(* IEC 61131-3 sources: elnaProjects/ElpcLogic/PomarKc7Changed/FunctionBlocks (part 2) *)

(* ---- Если управление с ВУ заблокировано, то  передаем команду из алгоритма ---- *)
IF StrAlg.inOpcCommandsDisabled THEN
	StrAlg.inCommand := StrAlg.inCommand_Alg;
ELSE (* иначе передаем команду с АРМа*)
	StrAlg.inCommand := StrAlg.inCommand_ARM;
END_IF;

_sunpackerCommand(command := StrAlg.inCommand);
	source := _sunpackerCommand.source;
	cmd := _sunpackerCommand.cmd;

IF cmd <> 0 AND lastCmd <> cmd AND (((NOT StrAlg.opcCommandsDisabled) AND source > 0) OR source = 0) then
	CASE BYTE_TO_INT(cmd) OF
		(*cmdRun*) 1: 	IF (StrAlg.CanRun) THEN
					StrAlg.isRuning := TRUE;
					StrAlg.isEnded := FALSE;
					StrAlg.hasError := FALSE;
					(*****************       OnRun       *****************)

					cmd_for_Status := cmd;
					source_for_Status := source;
					command_error_for_Status := 0;
				ELSE
					StrAlg.isRuning := FALSE;
					StrAlg.isEnded := FALSE;
					StrAlg.hasError 	:= FALSE;

					cmd_for_Status := 0;
					source_for_Status := source;
					command_error_for_Status := cmd;
				END_IF;
		(*cmdReset*) 2: 	StrAlg.isRuning := FALSE;
				StrAlg.isEnded := FALSE;
				StrAlg.hasError 	:= FALSE;

                                         (*****************       OnReset       *****************)
                                        waitOn(in:=FALSE);
                                        waitOff(in:=FALSE);
                                        AlgTimers.AutoPns_OffTimer:=UDINT_TO_UINT(TIME_TO_UDINT(waitOff.pt -waitOff.ET)/1000);

				cmd_for_Status := cmd;
				source_for_Status := source;
				command_error_for_Status := 0;
	END_CASE;
	resetCmdTimer(IN := false);
	resetCmdTimerPriznak := TRUE;
END_IF;
lastCmd := cmd;

resetCmdTimer(IN := resetCmdTimerPriznak, PT := T#5S);
IF resetCmdTimer.Q THEN
	resetCmdTimerPriznak := FALSE;
	source_for_Status := 0;
	cmd_for_Status := 0;
	command_error_for_Status := 0;
END_IF;

(*TODO: TYPE PROGRAM CODE HERE*)
StrAlg.status :=  SHL(BYTE_TO_DWORD(source_for_Status), 29)
			OR SHL(BYTE_TO_DWORD(cmd_for_Status), 26)
			OR SHL(BYTE_TO_DWORD(command_error_for_Status), 23)
			OR SHL(BOOL_TO_DWORD(StrAlg.OpcCommandsDisabled ), 21)
			OR SHL(BOOL_TO_DWORD(StrAlg.hasError),4)
			OR SHL(BOOL_TO_DWORD(StrAlg.CanRun),2)
			OR SHL(BOOL_TO_DWORD(StrAlg.isEnded),1)
			OR BOOL_TO_DWORD(StrAlg.isRuning);

(* ---- fb_AutoTenAlg.st ---- *)
FUNCTION_BLOCK fb_AutoTenAlg

VAR_IN_OUT
	StrAlg : struct_Alg;
	PNS : struct_Switch;
	TEN : struct_Switch;
END_VAR

VAR_INPUT
	T_masla : struct_AI;
	Uroven_masla : struct_AI;
	offTemperature : struct_AnalogParametr;
END_VAR

VAR
	_sunpackerCommand : fb_sunpackerCommand;
	_statusAi : TYPE_StatusAi;
	_statusDualInput : TYPE_statusDualInput;
	_commandDualInput : TYPE_commandDualInput;
	source : BYTE;
	cmd : BYTE;
	lastCmd : BYTE;
	source_for_Status : BYTE;
	cmd_for_Status : BYTE;
	command_error_for_Status : BYTE;
	resetCmdTimer : TON;
	resetCmdTimerPriznak : BOOL;
	onInit : BOOL;
END_VAR

IF NOT onInit THEN
StrAlg.inCanRun:=TRUE;
onInit:=TRUE;
END_IF;

IF StrAlg.isRuning THEN

IF ((T_masla.interval >= _statusAi.normal) AND (T_masla.value > offTemperature.Value)) OR
((Uroven_masla.interval >= _statusAi.normal) AND (Uroven_masla.value < Uroven_masla.LA)) OR
(PNS.onStatus=_statusDualInput.STATUS_OFF) THEN

      TEN.inOpcCommandsDisabled:=TRUE;

	IF TEN.onStatus = _statusDualInput.STATUS_ON THEN
          TEN.inCommand_Alg:=BYTE_TO_WORD(_commandDualInput.CMD_OFF);
	END_IF;

ELSIF PNS.onStatus = _statusDualInput.STATUS_ON THEN
      TEN.inOpcCommandsDisabled:=FALSE;
END_IF;

END_IF;

StrAlg.CanRun := StrAlg.inCanRun;
StrAlg.hasError := TEN.CommandFault OR (T_masla.interval < _statusAi.normal) OR (Uroven_masla.interval < _statusAi.normal);

StrAlg.OpcCommandsDisabled := StrAlg.inOpcCommandsDisabled;

(* ---- Если управление с ВУ заблокировано, то  передаем команду из алгоритма ---- *)
IF StrAlg.inOpcCommandsDisabled THEN
	StrAlg.inCommand := StrAlg.inCommand_Alg;
ELSE (* иначе передаем команду с АРМа*)
	StrAlg.inCommand := StrAlg.inCommand_ARM;
END_IF;

_sunpackerCommand(command := StrAlg.inCommand);
	source := _sunpackerCommand.source;
	cmd := _sunpackerCommand.cmd;

IF cmd <> 0 AND lastCmd <> cmd AND (((NOT StrAlg.opcCommandsDisabled) AND source > 0) OR source = 0) then
	CASE BYTE_TO_INT(cmd) OF
		(*cmdRun*) 1: 	IF StrAlg.CanRun AND NOT StrAlg.hasError THEN
					StrAlg.isRuning := TRUE;
					StrAlg.isEnded := FALSE;
					(*StrAlg.hasError := FALSE;*)

                                                  (*****************       OnRun       *****************)
                                                  IF StrAlg.inOpcCommandsDisabled THEN
		                              StrAlg.inOpcCommandsDisabled:=FALSE;
                                                  END_IF;
					cmd_for_Status := cmd;
					source_for_Status := source;
					command_error_for_Status := 0;
				ELSE
					StrAlg.isRuning := FALSE;
					StrAlg.isEnded := FALSE;
					(*StrAlg.hasError 	:= FALSE;*)

					cmd_for_Status := 0;
					source_for_Status := source;
					command_error_for_Status := cmd;
				END_IF;
		(*cmdReset*) 2: 	StrAlg.isRuning := FALSE;
				StrAlg.isEnded := FALSE;
				(*StrAlg.hasError 	:= FALSE;*)

                                        (*****************       OnReset       *****************)
                                        TEN.inOpcCommandsDisabled:=TRUE;
                                        TEN.inCommand_Alg:=BYTE_TO_WORD(_commandDualInput.CMD_OFF);

				cmd_for_Status := cmd;
				source_for_Status := source;
				command_error_for_Status := 0;
	END_CASE;
	resetCmdTimer(IN := false);
	resetCmdTimerPriznak := TRUE;
END_IF;
lastCmd := cmd;

resetCmdTimer(IN := resetCmdTimerPriznak, PT := T#5S);
IF resetCmdTimer.Q THEN
	resetCmdTimerPriznak := FALSE;
	source_for_Status := 0;
	cmd_for_Status := 0;
	command_error_for_Status := 0;
END_IF;

(*TODO: TYPE PROGRAM CODE HERE*)
StrAlg.status :=  SHL(BYTE_TO_DWORD(source_for_Status), 29)
			OR SHL(BYTE_TO_DWORD(cmd_for_Status), 26)
			OR SHL(BYTE_TO_DWORD(command_error_for_Status), 23)
			OR SHL(BOOL_TO_DWORD(StrAlg.OpcCommandsDisabled ), 21)
			OR SHL(BOOL_TO_DWORD(StrAlg.hasError),4)
			OR SHL(BOOL_TO_DWORD(StrAlg.CanRun),2)
			OR SHL(BOOL_TO_DWORD(StrAlg.isEnded),1)
			OR BOOL_TO_DWORD(StrAlg.isRuning);

(* ---- fb_BaseAlgoritm.st ---- *)
FUNCTION_BLOCK fb_BaseAlgoritm

VAR_IN_OUT
	StrAlg : struct_Alg;
END_VAR

VAR
	_sunpackerCommand : fb_sunpackerCommand;
	source : BYTE;
	cmd : BYTE;
	lastCmd : BYTE;
	source_for_Status : BYTE;
	cmd_for_Status : BYTE;
	command_error_for_Status : BYTE;
	resetCmdTimer : TON;
	resetCmdTimerPriznak : BOOL;
END_VAR

StrAlg.CanRun := StrAlg.inCanRun;
StrAlg.hasError := StrAlg.inHasError OR (command_error_for_Status <> 0);
StrAlg.isEnded := StrAlg.inEnded;

StrAlg.OpcCommandsDisabled := StrAlg.inOpcCommandsDisabled;

(* ---- Если управление с ВУ заблокировано, то передаем команду из алгоритма ---- *)
IF StrAlg.inOpcCommandsDisabled THEN
	StrAlg.inCommand := StrAlg.inCommand_Alg;
ELSE (* иначе передаем команду с АРМа*)
	StrAlg.inCommand := StrAlg.inCommand_ARM;
END_IF;

_sunpackerCommand(command := StrAlg.inCommand);
	source := _sunpackerCommand.source;
	cmd := _sunpackerCommand.cmd;

IF cmd <> 0 AND lastCmd <> cmd AND (((NOT StrAlg.opcCommandsDisabled) AND source > 0) OR source = 0) then
	CASE BYTE_TO_INT(cmd) OF
		(*cmdRun*) 1: 	IF (StrAlg.CanRun) THEN
					StrAlg.isRuning := TRUE;
					StrAlg.isEnded := FALSE;
					StrAlg.hasError 	:= FALSE;

					cmd_for_Status := cmd;
					source_for_Status := source;
					command_error_for_Status := 0;
				ELSE
					StrAlg.isRuning := FALSE;
					StrAlg.isEnded := FALSE;
					StrAlg.hasError 	:= FALSE;

					cmd_for_Status := 0;
					source_for_Status := source;
					command_error_for_Status := cmd;
				END_IF;
		(*cmdReset*) 2: 	StrAlg.isRuning := FALSE;
				StrAlg.isEnded := FALSE;
				StrAlg.hasError 	:= FALSE;
				cmd_for_Status := cmd;
				source_for_Status := source;
				command_error_for_Status := 0;
	END_CASE;
	resetCmdTimer(IN := false);
	resetCmdTimerPriznak := TRUE;
END_IF;
lastCmd := cmd;

resetCmdTimer(IN := resetCmdTimerPriznak, PT := T#5S);
IF resetCmdTimer.Q THEN
	resetCmdTimerPriznak := FALSE;
	source_for_Status := 0;
	cmd_for_Status := 0;
	command_error_for_Status := 0;
END_IF;

StrAlg.status :=  SHL(BYTE_TO_DWORD(source_for_Status), 29)
			OR SHL(BYTE_TO_DWORD(cmd_for_Status), 26)
			OR SHL(BYTE_TO_DWORD(command_error_for_Status), 23)
			OR SHL(BOOL_TO_DWORD(StrAlg.OpcCommandsDisabled ), 21)
			OR SHL(BOOL_TO_DWORD(StrAlg.hasError),4)
			OR SHL(BOOL_TO_DWORD(StrAlg.CanRun),2)
			OR SHL(BOOL_TO_DWORD(StrAlg.isEnded),1)
			OR BOOL_TO_DWORD(StrAlg.isRuning);

(* ---- fb_BaseProtection.st ---- *)
FUNCTION_BLOCK fb_BaseProtection

VAR_INPUT
	inSignaling : BOOL;
	inTag : BYTE;
	inRunOnStart : BOOL;
	inCanRun : BOOL;
	inHasError : BOOL;
	inEnded : BOOL;
	inOpcCommandsDisabled : BOOL;
	inCommand : WORD;
END_VAR

VAR_OUTPUT
	Tag : BYTE;
	status : DWORD;
	CanRun : BOOL;
	OpcCommandsDisabled : BOOL;
	isRunning : BOOL;
	HasError : BOOL;
	isEnded : BOOL;
	Remont : BOOL;
	Check : BOOL;
	Signaling : BOOL;
	SignalingTP : BOOL;
	RunOnStart : BOOL;
END_VAR

VAR
	_sunpackerCommand : fb_sunpackerCommand;
	_ProtectionTags : TYPE_ProtectionTags;
	_signalingTp : TOF;
	source : BYTE;
	cmd : BYTE;
	lastCmd : BYTE;
	source_for_Status : BYTE;
	cmd_for_Status : BYTE;
	command_error_for_Status : BYTE;
	resetCmdTimer : TON;
	resetCmdTimerPriznak : BOOL;
	signalinTimer : TON;
	runOnStart_Trig : R_TRIG;
END_VAR

Tag := inTag;
RunOnStart := inRunOnStart;

CanRun := inCanRun;
hasError := inHasError;
isEnded := inEnded;

OpcCommandsDisabled := inOpcCommandsDisabled;

_sunpackerCommand(command := inCommand);
	source := _sunpackerCommand.source;
	cmd := _sunpackerCommand.cmd;

IF cmd <> 0 AND lastCmd <> cmd AND (((NOT opcCommandsDisabled) AND source > 0) OR source = 0) then
	CASE BYTE_TO_INT(cmd) OF
		(*cmdRun*) 1: 	IF CanRun AND NOT Remont THEN
					isEnded := FALSE;
					hasError 	:= FALSE;
					isRunning := TRUE;
					cmd_for_Status := cmd;
					source_for_Status := source;
					command_error_for_Status := 0;
				ELSE
					isRunning := FALSE;
					isEnded := FALSE;
					hasError 	:= FALSE;

					cmd_for_Status := 0;
					source_for_Status := source;
					command_error_for_Status := cmd;
				END_IF;
		(*cmdReset*) 2: 	isRunning := FALSE;
				isEnded := FALSE;
				hasError 	:= FALSE;
				inSignaling := FALSE;
				Check := FALSE;
				cmd_for_Status := cmd;
				source_for_Status := source;
				command_error_for_Status := 0;
	(*cmd_setRemont*) 4 :	Remont := TRUE;
				isRunning := FALSE;

				cmd_for_Status := cmd;
				source_for_Status := source;
				command_error_for_Status := 0;
	(*cmd_resetRemont*) 5 : 	IF inSignaling THEN
					cmd_for_Status := 0;
					source_for_Status := 0;
					command_error_for_Status := cmd;
				ELSE
					Remont := FALSE;
					isRunning := TRUE;

					cmd_for_Status := cmd;
					source_for_Status := source;
					command_error_for_Status := 0;
				END_IF;
	(*cmd_setCheck*) 6 : 	Check := TRUE;

				cmd_for_Status := cmd;
				source_for_Status := source;
				command_error_for_Status := 0;
	END_CASE;
	resetCmdTimer(IN := false);
	resetCmdTimerPriznak := TRUE;
END_IF;
lastCmd := cmd;

resetCmdTimer(IN := resetCmdTimerPriznak);
IF resetCmdTimer.Q THEN
	resetCmdTimerPriznak := FALSE;
	source_for_Status := 0;
	cmd_for_Status := 0;
	command_error_for_Status := 0;
END_IF;

IF isRunning THEN
	Signaling := inSignaling;
	SignalingTP := _signalingTp.Q;
ELSE
	Signaling := 0;
	SignalingTP := 0;
END_IF;

IF NOT Remont AND NOT Check THEN
	_signalingTp(in := Signaling, PT := T#1s);
ELSE
	_signalingTp(in := FALSE);
END_IF;

status :=  SHL(BYTE_TO_DWORD(source_for_Status), 29)
			OR SHL(BYTE_TO_DWORD(cmd_for_Status), 26)
			OR SHL(BYTE_TO_DWORD(command_error_for_Status), 23)
			OR SHL(BOOL_TO_DWORD(OpcCommandsDisabled ), 21)
			OR SHL(BOOL_TO_DWORD(Signaling), 16)
			OR SHL(BOOL_TO_DWORD(RunOnStart ), 15)
			OR SHL(BOOL_TO_DWORD(remont), 6)
			OR SHL(BOOL_TO_DWORD(Check), 5)
			OR SHL(BOOL_TO_DWORD(hasError), 4)
			OR SHL(BOOL_TO_DWORD(SignalingTP), 3)
			OR SHL(BOOL_TO_DWORD(CanRun), 2)
			OR SHL(BOOL_TO_DWORD(isEnded), 1)
			OR BOOL_TO_DWORD(isRunning);

(* ---- fb_DI_Init.st ---- *)
FUNCTION_BLOCK fb_DI_Init

VAR_INPUT
	data_Ini : BOOL; (*Флаг необходимости инициализации параметров.*)
	imit : BOOL          := FALSE;
END_VAR

VAR_IN_OUT
	strDI : struct_DI;
END_VAR

VAR_OUTPUT
	Init : BOOL          := FALSE; (*Флаг успешно выполненной инициализации.*)
END_VAR

(*****            Функциональный блок переинициализации структуры-дескриптора канала дискретного ввода        *****)

 Init := FALSE;

    IF data_Ini THEN                            (* Параметрам требуется переинициализация. *)
        strDI.imit       := imit;
        data_Ini:=FALSE;
        Init := TRUE;
    END_IF;
  IF Init THEN
imit:=FALSE;
    END_IF;

(* ---- fb_DiProtection.st ---- *)
FUNCTION_BLOCK fb_DiProtection

VAR_INPUT
	di : struct_singleSignal;
END_VAR

VAR_IN_OUT
	StrDIp : struct_DiProtection;
END_VAR

VAR
	_sunpackerCommand : fb_sunpackerCommand;
	_ProtectionTags : TYPE_ProtectionTags;
	_signalingTp : TOF;
	timer : TON;
	SignalingTrig : R_TRIG;
	SignalingFTrig : F_TRIG;
	SignalingDi : BOOL;
	source : BYTE;
	cmd : BYTE;
	lastCmd : BYTE;
	source_for_Status : BYTE;
	cmd_for_Status : BYTE;
	command_error_for_Status : BYTE;
	resetCmdTimer : TON;
	resetCmdTimerPriznak : BOOL;
	signalinTimer : TON;
	runOnStart_Trig : R_TRIG;
END_VAR

timer(IN := di.Q AND StrDIp.isRunning  , PT := StrDIp.delay);
SignalingTrig(CLK := timer.Q);
IF SignalingTrig.Q THEN
	SignalingDi := TRUE;
END_IF;
SignalingFTrig(CLK := timer.Q);
IF SignalingFTrig.Q THEN
	SignalingDi := FALSE;
END_IF;

StrDIp.Tag := StrDIp.inTag;
StrDIp.RunOnStart := StrDIp.inRunOnStart;

StrDIp.CanRun := StrDIp.inCanRun;

StrDIp.OpcCommandsDisabled := StrDIp.inOpcCommandsDisabled;

(* ---- Если управление с ВУ заблокировано, то передаем команду из алгоритма ---- *)
IF StrDIp.inOpcCommandsDisabled THEN
	StrDIp.inCommand := StrDIp.inCommand_Alg;
ELSE (* иначе передаем команду с АРМа*)
	StrDIp.inCommand := StrDIp.inCommand_ARM;
END_IF;

_sunpackerCommand(command := StrDIp.inCommand);
	source := _sunpackerCommand.source;
	cmd := _sunpackerCommand.cmd;

IF cmd <> 0 AND lastCmd <> cmd AND (((NOT StrDIp.opcCommandsDisabled) AND source > 0) OR source = 0) then

	CASE BYTE_TO_INT(cmd) OF
	        (*cmdRun*) 1: 	IF        NOT StrDIp.Remont THEN
					StrDIp.isEnded := FALSE;
					StrDIp.hasError 	:= FALSE;
					StrDIp.isRunning := TRUE;
					cmd_for_Status := cmd;
					source_for_Status := source;
					command_error_for_Status := 0;
				ELSE
					StrDIp.isRunning := FALSE;
					StrDIp.isEnded := FALSE;
					StrDIp.hasError 	:= FALSE;

					cmd_for_Status := 0;
					source_for_Status := source;
					command_error_for_Status := cmd;
				END_IF;
                                        StrDIp.inOpcCommandsDisabled:=FALSE;

                (*cmdReset*) 2: 	StrDIp.isRunning := FALSE;
				StrDIp.isEnded := FALSE;
				StrDIp.hasError 	:= FALSE;
				SignalingDi:= FALSE;
				StrDIp.Check := FALSE;
				cmd_for_Status := cmd;
				source_for_Status := source;
				command_error_for_Status := 0;
                                       StrDIp.inOpcCommandsDisabled:=FALSE;

	(*cmd_setRemont*) 4 :	StrDIp.Remont := TRUE;
				(*StrDIp.isRunning := FALSE;*)

				cmd_for_Status := cmd;
				source_for_Status := source;
				command_error_for_Status := 0;
        (*cmd_resetRemont*) 5 : 	(*IF di.Q THEN
					cmd_for_Status := 0;
					source_for_Status := 0;
					command_error_for_Status := cmd;
				ELSE*)
					StrDIp.Remont := FALSE;
					(*StrDIp.isRunning := TRUE;*)

					cmd_for_Status := cmd;
					source_for_Status := source;
					command_error_for_Status := 0;
				(*END_IF;*)
	(*cmd_setCheck*) 6 : 	StrDIp.Check := TRUE;

				cmd_for_Status := cmd;
				source_for_Status := source;
				command_error_for_Status := 0;
	END_CASE;
	resetCmdTimer(IN := false);
	resetCmdTimerPriznak := TRUE;
END_IF;
lastCmd := cmd;

resetCmdTimer(IN := resetCmdTimerPriznak);
IF resetCmdTimer.Q THEN
	resetCmdTimerPriznak := FALSE;
	source_for_Status := 0;
	cmd_for_Status := 0;
	command_error_for_Status := 0;
END_IF;

IF StrDIp.isRunning AND NOT StrDIp.Remont AND NOT StrDIp.Check THEN
	StrDIp.Signaling := SignalingDi;
	StrDIp.SignalingTP := _signalingTp.Q;
ELSE
	StrDIp.Signaling := 0;
	StrDIp.SignalingTP := 0;
END_IF;

_signalingTp(in := StrDIp.Signaling, PT := T#1s);

StrDIp.status :=  SHL(BYTE_TO_DWORD(source_for_Status), 29)
			OR SHL(BYTE_TO_DWORD(cmd_for_Status), 26)
			OR SHL(BYTE_TO_DWORD(command_error_for_Status), 23)
			OR SHL(BOOL_TO_DWORD(StrDIp.OpcCommandsDisabled ), 21)
			OR SHL(BOOL_TO_DWORD(StrDIp.Signaling), 16)
			OR SHL(BOOL_TO_DWORD(StrDIp.RunOnStart ), 15)
			OR SHL(BOOL_TO_DWORD(StrDIp.remont), 6)
			OR SHL(BOOL_TO_DWORD(StrDIp.Check), 5)
			OR SHL(BOOL_TO_DWORD(StrDIp.hasError), 4)
			OR SHL(BOOL_TO_DWORD(StrDIp.SignalingTP), 3)
			OR SHL(BOOL_TO_DWORD(StrDIp.CanRun), 2)
			OR SHL(BOOL_TO_DWORD(StrDIp.isEnded), 1)
			OR BOOL_TO_DWORD(StrDIp.isRunning);

(* ---- fb_DiProtection_Init.st ---- *)
FUNCTION_BLOCK fb_DiProtection_Init

VAR_INPUT
	data_Ini : BOOL; (*Флаг необходимости инициализации параметров.*)
	delay : TIME;
	inTag : BYTE;
	inRunOnStart : BOOL;
END_VAR

VAR_IN_OUT
	str_DIp : struct_DiProtection;
END_VAR

VAR_OUTPUT
	Init : BOOL          := FALSE; (*Флаг успешно выполненной инициализации.*)
END_VAR

(*****            Функциональный блок переинициализации структуры  AiProtection          *****)

 Init := FALSE;

    IF data_Ini THEN                            (* Параметрам требуется переинициализация. *)
        str_DIp.delay               := delay;
        str_DIp.inTag               := inTag;
        str_DIp.inRunOnStart        := inRunOnStart;

        data_Ini:=FALSE;
        Init := TRUE;
    END_IF;
    IF Init THEN
        delay:= T#0S;
        inTag:= 0;
        inRunOnStart:= FALSE;
    END_IF;

(* ---- fb_DiscretParametr.st ---- *)
FUNCTION_BLOCK fb_DiscretParametr

VAR_IN_OUT
	StrDP : struct_DiscretParametr;
END_VAR

VAR
	_sunpackerCommand : fb_sunpackerCommand;
	source : BYTE;
	cmd : BYTE;
	parametr : BYTE;
	lastParametr : BYTE;
	source_for_Status : BYTE;
	cmd_for_Status : BYTE;
	command_error_for_Status : BYTE;
	resetCmdTimer : TON;
	resetCmdTimerPriznak : BOOL;
	secondTact : BOOL;
END_VAR

IF NOT secondTact THEN
	StrDP.Value := StrDP.currentValue;
	secondTact := true;
END_IF;

StrDP.OpcCommandsDisabled := StrDP.inOpcCommandsDisabled;

(* ---- Если управление с ВУ заблокировано, то передаем команду из алгоритма ---- *)
IF StrDP.inOpcCommandsDisabled THEN
	StrDP.inCommand := StrDP.inCommand_Alg;
ELSE (* иначе передаем команду с АРМа*)
	StrDP.inCommand := StrDP.inCommand_ARM;
END_IF;

_sunpackerCommand(command := StrDP.inCommand);
	source := _sunpackerCommand.source;
          parametr := _sunpackerCommand.parametr;
	cmd := _sunpackerCommand.cmd;

IF NOT StrDP.inOpcCommandsDisabled THEN
StrDP.newValue:= BYTE_TO_UINT(parametr);
END_IF;

IF cmd <> 0 AND StrDP.Value <> StrDP.newValue AND (((NOT StrDP.opcCommandsDisabled) AND source > 0) OR source = 0) then
	CASE BYTE_TO_INT(cmd) OF
	(*cmd_ChangeValue*) 1 :
                                  StrDP.Value := StrDP.newValue;
                                  StrDP.opcCommandsDisabled:=FALSE;
	END_CASE;
	source_for_Status := source;
	cmd_for_Status := cmd;
	resetCmdTimer(IN := FALSE);
	resetCmdTimerPriznak := TRUE;
END_IF;

lastParametr := parametr;

StrDP.status := SHL(BYTE_TO_DWORD(source_for_Status), 29)
			OR SHL(BYTE_TO_DWORD(cmd_for_Status), 26)
			OR SHL(BYTE_TO_DWORD(command_error_for_Status), 23)
			OR SHL(BOOL_TO_DWORD(StrDP.OpcCommandsDisabled ), 21)
                              OR SHL(UINT_TO_DWORD(StrDP.Value), 5);

resetCmdTimer(IN := resetCmdTimerPriznak, PT := T#5S);
IF resetCmdTimer.Q THEN
	resetCmdTimerPriznak := FALSE;
	source_for_Status := 0;
	cmd_for_Status := 0;
	command_error_for_Status := 0;
END_IF;

(* ---- fb_DiscretParametr_Init.st ---- *)
FUNCTION_BLOCK fb_DiscretParametr_Init

VAR_INPUT
	data_Ini : BOOL; (*Флаг необходимости инициализации параметров.*)
	currentValue : UINT;
END_VAR

VAR_IN_OUT
	strDp : struct_DiscretParametr;
END_VAR

VAR_OUTPUT
	Init : BOOL          := FALSE; (*Флаг успешно выполненной инициализации.*)
END_VAR

(*****            Функциональный блок переинициализации дискретного параметра.          *****)

 Init := FALSE;

    IF data_Ini THEN                            (* Параметрам требуется переинициализация. *)
        strDp.currentValue       := currentValue;
        data_Ini:=FALSE;
        Init := TRUE;
    END_IF;
IF Init THEN
currentValue:=0;
END_IF;

(* ---- fb_DiSourceMlp.st ---- *)
FUNCTION_BLOCK fb_DiSourceMlp

VAR_INPUT
	arDIN : TItemDIN;
	err_mod : TItemDIN;
END_VAR

VAR_IN_OUT
	strDI : struct_DI;
END_VAR

VAR_OUTPUT
	Bounce : BOOL; (*Дребезг контактов*)
END_VAR

VAR
	_value : WORD;
	_reliability : BOOL;
	bitNumber : INT;
	bitNum : INT;
END_VAR

strDI.blConnect := (*((UINT_TO_WORD(arDIN.wFlags) = 1472) and*) (UINT_TO_WORD(err_mod.wValue) = 20) and (UINT_TO_WORD(err_mod.wFlags) = 192);
Bounce := (UINT_TO_WORD(arDIN.wFlags) AND 16#0020) <> 0;

If NOT strDI.imit THEN
_value:=UINT_TO_WORD(arDIN.wValue);

    IF strDI.blConnect THEN
          strDI.reliability:=0;
          strDI.value:=0;
	FOR bitNumber:=0 TO 7 BY 1 DO

		_reliability:=WORD_TO_BOOL(SHR(_value, bitNumber*2) AND 16#2);
		strDI.reliability:=strDI.reliability OR SHL(BOOL_TO_WORD(_reliability),bitNumber);
		IF _reliability THEN
			strDI.value:=strDI.value OR SHL((SHR(_value, bitNumber*2) AND 16#1),bitNumber);
		END_IF;
	END_FOR;
    ELSE
	strDI.reliability := 0;
    END_IF;

    FOR bitNum:=0 TO 15 BY 1 DO
	          strDI.bits[bitNum].reliability :=WORD_TO_BOOL(SHR(strDI.reliability, bitNum) AND 16#1);
	IF strDI.bits[bitNum].reliability THEN
		strDI.bits[bitNum].value :=WORD_TO_BOOL(SHR(strDI.value, bitNum) AND 16#1);
                    strDI.bits[bitNum]._inversed :=NOT strDI.bits[bitNum].value;
	END_IF;
    END_FOR;

END_IF;

(* ---- fb_DO_Init.st ---- *)
FUNCTION_BLOCK fb_DO_Init

VAR_INPUT
	data_Ini : BOOL; (*Флаг необходимости инициализации параметров.*)
	imit : BOOL          := FALSE; (*Действие при неисправности канала AI.*)
END_VAR

VAR_IN_OUT
	strDO : struct_DO; (*Дескриптор DO-канала.*)
END_VAR

VAR_OUTPUT
	Init : BOOL          := FALSE; (*Флаг успешно выполненной инициализации.*)
END_VAR

(*****            Функциональный блок переинициализации структуры-дескриптора канала дискретного ввода.            *****)
 Init := FALSE;

    IF data_Ini THEN                            (* Параметрам требуется переинициализация. *)
        strDO.imit       := imit;
        data_Ini:=FALSE;
        Init := TRUE;
    END_IF;
  IF Init THEN
imit:=FALSE;
   END_IF;

(* ---- fb_DOSourceMlp.st ---- *)
FUNCTION_BLOCK fb_DOSourceMlp

VAR_IN_OUT
	arDout : TWordData; (*Данные для модуля DO.*)
END_VAR

VAR_INPUT
	err_mod : TItemDIN;
END_VAR

VAR_IN_OUT
	strDO : struct_DO; (*Текущие параметры канала DO.*)
END_VAR

VAR
	bitNumber : INT;
END_VAR

strDO.blConnect := ((UINT_TO_WORD(err_mod.wValue) = 20) and (UINT_TO_WORD(err_mod.wFlags) = 192));

strDO.value:=0;

FOR bitNumber:=0 TO 15 BY 1 DO
	strDO.value:=strDO.value OR (SHL(BOOL_TO_WORD(strDO.bits[bitNumber]),bitNumber));
END_FOR;

IF NOT strDO.imit THEN
	 arDout.wValue:= WORD_TO_UINT(strDO.value);
END_IF;

(* ---- fb_DualStateIm.st ---- *)
FUNCTION_BLOCK fb_DualStateIm

VAR_INPUT
	statOn : BOOL;
	statOff : BOOL;
END_VAR

VAR_IN_OUT
	StrDs : struct_DualStateIm;
END_VAR

VAR_INPUT
	statOn_reliability : BOOL;
	statOff_reliability : BOOL;
	inNs : TYPE_ReliableBit;
	inAccident : TYPE_ReliableBit;
	inCommand : WORD;
END_VAR

VAR
	_statOn : BOOL;
	_statOff : BOOL;
	getSdvig : BOOL;
	lastOnStatus : BYTE;
	cmd : BYTE;
	source : BYTE;
	lastCmd : BYTE;
	source_for_Status : BYTE;
	cmd_for_Status : BYTE;
	command_error_for_Status : BYTE;
	_sunpackerCommand : fb_sunpackerCommand;
	_statusDualInput : TYPE_statusDualInput;
	_commandDualInput : TYPE_commandDualInput;
	_commandErrorTimer : BOOL;
	onInit : BOOL          := FALSE;
	resetErrorTimer : BOOL;
	_changWithoutCommand : BOOL;
	errorCMDTimer : TON;
	sdvigReset : TON;
	_errorReset : TON;
END_VAR

VAR_IN_OUT
	cmdOn : BOOL;
END_VAR

VAR_OUTPUT
	cmdOff : BOOL;
END_VAR

IF NOT onInit THEN
IF StrDs.ISVALIDREF_cmdOn XOR StrDs.ISVALIDREF_cmdOff THEN
	IF 	StrDs.ISVALIDREF_cmdOn THEN
		lastCmd:= 2; (*baseCmdOff*)
	ELSE
		lastCmd:= 1; (*baseCmdOn*)
	END_IF;
END_IF;
onInit:=TRUE;
END_IF;

(* ---- Если управление с ВУ заблокировано, то в ИМ передаем команду из алгоритма ---- *)
IF StrDs.inOpcCommandsDisabled THEN
	StrDs.inCommand := StrDs.inCommand_Alg;
ELSE (* иначе передаем команду с АРМа*)
	StrDs.inCommand := StrDs.inCommand_ARM;
END_IF;

(* ---- Формирование состояния механизма ---- *)

IF (StrDs.ISVALIDREF_statOn) OR (StrDs.ISVALIDREF_statOff) THEN
	IF (StrDs.ISVALIDREF_statOn) AND (StrDs.ISVALIDREF_statOff) THEN
	StrDs.reliability:= statOn_reliability AND statOff_reliability;
		_statOn  := statOn;
		_statOff := statOff;
	ELSIF (StrDs.ISVALIDREF_statOn) THEN
                     StrDs.reliability:= statOn_reliability;
		_statOn  := statOn;
		_statOff := NOT statOn;
	ELSIF (StrDs.ISVALIDREF_statOff) THEN
		 StrDs.reliability:= statOff_reliability;
		_statOn  := NOT statOff;
		_statOff :=statOff;
	END_IF;

	IF StrDs.reliability THEN
		IF _statOn AND NOT _statOff 		THEN 	StrDs.onStatus := _statusDualInput.STATUS_ON;
		ELSIF _statOff AND NOT _statOn 	THEN 	StrDs.onStatus := _statusDualInput.Status_OFF;
		ELSIF NOT _statOn AND NOT _statOff 	THEN 	StrDs.onStatus := _statusDualInput.STATUS_TRANSITIONAL;
		ELSE					StrDs.onStatus := _statusDualInput.STATUS_ERROR;
                    END_IF;

	ELSE
		StrDs.onStatus := _statusDualInput.STATUS_NOTDEFINED;

	END_IF;
ELSE
	CASE BYTE_TO_INT(lastCmd) OF
		(*baseCmdOn*) 1: StrDs.onStatus  := _statusDualInput.STATUS_ON;
		(*baseCmdOff*) 2: StrDs.onStatus  := _statusDualInput.STATUS_OFF;

	ELSE
		 StrDs.onStatus := _statusDualInput.STATUS_NOTDEFINED;

	END_CASE;
END_IF;

(* ---- Формирование признака сдвига ---- *)
getSdvig := FALSE;
IF (StrDs.ISVALIDREF_cmdOn OR StrDs.ISVALIDREF_cmdOff) THEN
	IF NOT (StrDs.CmdOn OR StrDs.CmdOff) THEN
                     IF (lastOnStatus <> StrDs.onStatus AND
		(StrDs.onStatus <> _statusDualInput.STATUS_NOTDEFINED AND
                     StrDs.onStatus <> _statusDualInput.STATUS_ERROR)     AND
		(lastOnStatus <> _statusDualInput.STATUS_NOTDEFINED   AND
                     lastOnStatus <> _statusDualInput.STATUS_ERROR))
                    THEN
			getSdvig   := TRUE;
		END_IF;
	END_IF;
END_IF;

IF getSdvig THEN StrDs.sdvig:= TRUE; END_IF;

sdvigReset(IN:=StrDs.sdvig, PT:=T#15S);

IF sdvigReset.Q THEN StrDs.sdvig:=FALSE; END_IF;

lastOnStatus := StrDs.onStatus;

StrDs.Accident := inAccident.value AND inAccident.reliability;
StrDs.Ns := inNs.value AND inNs.reliability;
StrDs.OpcCommandsDisabled := StrDs.inOpcCommandsDisabled;

(* ---- Распаковка команды ---- *)
_sunpackerCommand(command := StrDs.inCommand);
	cmd := _sunpackerCommand.cmd;
	source := _sunpackerCommand.source;

(* ---- Обработка команды ---- *)
IF cmd <> 0 AND lastCmd <> cmd and (((NOT StrDs.opcCommandsDisabled) AND source > 0) OR source = 0) then
	CASE BYTE_TO_INT(cmd) OF
	(*cmd_open*) 1 :
			IF  StrDs.ISVALIDREF_cmdOn THEN StrDs.CmdOn := TRUE;
				IF StrDs.ISVALIDREF_cmdOff THEN StrDs.CmdOff := FALSE; END_IF;
			ELSIF  StrDs.ISVALIDREF_cmdOff THEN StrDs.CmdOff := FALSE;  END_IF;
			errorCMDTimer(IN := false);
			_commandErrorTimer := true;
			StrDs.lastCmdIsOn := true;
	(*cmd_close*) 2 :
			IF StrDs.ISVALIDREF_cmdOff THEN StrDs.CmdOff := TRUE;
				IF StrDs.ISVALIDREF_cmdOn THEN StrDs.CmdOn := FALSE; END_IF;
			ELSIF StrDs.ISVALIDREF_cmdOn THEN StrDs.CmdOn := FALSE; END_IF;
			errorCMDTimer(IN := false);
			_commandErrorTimer := true;
			StrDs.lastCmdIsOn := false;
	(*cmd_reset*) 3 :    IF StrDs.ISVALIDREF_statOn OR StrDs.ISVALIDREF_statOff THEN
			StrDs.CmdOn := FALSE;
			StrDs.CmdOff := FALSE;
                              lastCmd :=0;
			_commandErrorTimer := false;
			StrDs.lastCmdIsOn := false;
                              END_IF;
	END_CASE;
	source_for_Status := source;
	cmd_for_Status := cmd;
	command_error_for_Status := 0;
END_IF;

lastCmd := cmd;
errorCMDTimer(In := _commandErrorTimer, PT :=T#10s);

(* ---- алгоритм  для команды ВКЛючить ---- *)
IF (StrDs.onStatus = _statusDualInput.STATUS_ON) and (lastCmd = _commandDualInput.CMD_ON) then
	IF StrDs.ISVALIDREF_cmdOn AND StrDs.ISVALIDREF_cmdOff then  StrDs.cmdOn := false; END_IF;

	 errorCMDTimer(In := false);
	 _commandErrorTimer := false;
	 cmd_for_Status := 0;
	 source_for_Status := 0;
END_IF;

(* ---- off ---- *)
IF (StrDs.onStatus = _statusDualInput.STATUS_OFF) and (lastCmd = _commandDualInput.CMD_OFF) then
	IF StrDs.ISVALIDREF_cmdOn AND StrDs.ISVALIDREF_cmdOff then  StrDs.cmdOff := false; END_IF;

	 errorCMDTimer(In := false);
	 _commandErrorTimer := false;
	 cmd_for_Status := 0;
	 source_for_Status := 0;
END_IF;

(* ---- ошибка исполнения команды ---- *)
if errorCMDTimer.Q and (cmd_for_Status <> 0) then
	command_error_for_Status :=  cmd_for_Status;
	_commandErrorTimer := false;
	StrDs.CmdOn := false;
	StrDs.CmdOff := false;
	lastCmd := 0;
end_if;

(* ---- сброс ошибки команды ---- *)
StrDs.CommandFault := command_error_for_Status <> 0;
_errorReset(IN := command_error_for_Status <> 0, PT := T#15S);
IF _errorReset.Q THEN
	cmd_for_Status := 0;
	source_for_Status := 0;
	command_error_for_Status := 0;
END_IF;

cmdOn := StrDs.cmdOn;
cmdOff:= StrDs.cmdOff;

(* ---- формирование зашифрованного статуса для АРМа ---- *)
StrDs.status := shl(BYTE_TO_DWORD(source_for_Status), 29)
		OR shl(BYTE_TO_DWORD(cmd_for_Status), 26)
		OR shl(BYTE_TO_DWORD(command_error_for_Status), 23)
		OR shl(bool_to_DWORD(StrDs.sdvig), 22)
		OR shl(bool_to_DWORD(StrDs.OpcCommandsDisabled), 21)
		OR shl(BOOL_TO_DWORD(StrDs.Ns), 4)
                	OR shl(BOOL_TO_DWORD(StrDs.Accident ),3)
		OR BYTE_TO_DWORD(StrDs.onStatus);

(* ---- fb_Kran.st ---- *)
FUNCTION_BLOCK fb_Kran

VAR_INPUT
	statOn : BOOL;
	statOff : BOOL;
	statOn_reliability : BOOL;
	statOff_reliability : BOOL;
END_VAR

VAR_IN_OUT
	strKr : struct_Kran;
END_VAR

VAR_INPUT
	inNs : TYPE_ReliableBit;
	inAccident : TYPE_ReliableBit;
	inAuto : TYPE_ReliableBit;
	inManual : TYPE_ReliableBit;
	inLocal : TYPE_ReliableBit;
	inDistance : TYPE_ReliableBit;
	inErrorPowerOff : TYPE_ReliableBit;
	inErrorBlock : TYPE_ReliableBit;
	inSo : TYPE_ReliableBit;
	inSz : TYPE_ReliableBit;
	inDp : TYPE_ReliableBit;
END_VAR

VAR
	onInit : BOOL          := FALSE;
	_statOn : BOOL;
	_statOff : BOOL;
	getSdvig : BOOL;
	lastOnStatus : BYTE;
	cmd : BYTE;
	source : BYTE;
	lastCmd : BYTE;
	source_for_Status : BYTE;
	cmd_for_Status : BYTE;
	command_error_for_Status : BYTE;
	_sunpackerCommand : fb_sunpackerCommand;
	_statusDualInput : TYPE_statusDualInput;
	_commandDualInput : TYPE_commandDualInput;
	_commandErrorTimer : BOOL;
	resetErrorTimer : BOOL;
	_changWithoutCommand : BOOL;
	BlockedOpenControl : BOOL;
	errorCMDTimer : TON;
	_errorReset : TON;
	sdvigReset : TON;
	continueHoldCommandTimer : TON;
	outputsSets : TOF;
	dP_Trig : R_TRIG;
	dP_Trig_reliability : R_TRIG;
	resetBlockedOpenControl_Trig : R_TRIG;
END_VAR

VAR_IN_OUT
	cmdOn : BOOL;
	cmdOff : BOOL;
END_VAR

IF NOT onInit THEN
IF strKr.ISVALIDREF_cmdOn XOR strKr.ISVALIDREF_cmdOff THEN
	IF 	strKr.ISVALIDREF_cmdOn THEN
		lastCmd:= 2; (*baseCmdOff*)
	ELSE
		lastCmd:= 1; (*baseCmdOn*)
	END_IF;
END_IF;
onInit:=TRUE;
END_IF;

(* ---- Если управление с ВУ заблокировано, то в ИМ передаем команду из алгоритма ---- *)
IF strKr.inOpcCommandsDisabled THEN
	strKr.inCommand := strKr.inCommand_Alg;
ELSE (* иначе передаем команду с АРМа*)
	strKr.inCommand := strKr.inCommand_ARM;
END_IF;

(* ---- Формирование состояния механизма ---- *)

IF (strKr.ISVALIDREF_statOn) OR (strKr.ISVALIDREF_statOff) THEN
	IF (strKr.ISVALIDREF_statOn) AND (strKr.ISVALIDREF_statOff) THEN
	strKr.reliability:= statOn_reliability AND statOff_reliability;
		_statOn  := statOn;
		_statOff := statOff;
	ELSIF (strKr.ISVALIDREF_statOn) THEN
                     strKr.reliability:= statOn_reliability;
		_statOn  := statOn;
		_statOff := NOT statOn;
	ELSIF (strKr.ISVALIDREF_statOff) THEN
		 strKr.reliability:= statOff_reliability;
		_statOn  := NOT statOff;
		_statOff :=statOff;
	END_IF;

	IF strKr.reliability THEN
		IF _statOn AND NOT _statOff 		THEN 	strKr.onStatus := _statusDualInput.STATUS_ON;
		ELSIF _statOff AND NOT _statOn 	THEN 	strKr.onStatus := _statusDualInput.Status_OFF;
		ELSIF NOT _statOn AND NOT _statOff 	THEN 	strKr.onStatus := _statusDualInput.STATUS_TRANSITIONAL;
		ELSE					strKr.onStatus := _statusDualInput.STATUS_ERROR;
                    END_IF;

	ELSE
		strKr.onStatus := _statusDualInput.STATUS_NOTDEFINED;

	END_IF;
ELSE
	CASE BYTE_TO_INT(lastCmd) OF
		(*baseCmdOn*)  1: strKr.onStatus  := _statusDualInput.STATUS_ON;
		(*baseCmdOff*) 2: strKr.onStatus  := _statusDualInput.STATUS_OFF;

	ELSE
		 strKr.onStatus := _statusDualInput.STATUS_NOTDEFINED;

	END_CASE;
END_IF;

strKr.Accident := inAccident.value AND inAccident.reliability;
strKr.Ns := inNs.value AND inNs.reliability;
strKr.Auto := inAuto.value AND inAuto.reliability;
strKr.Manual := inManual.value AND inManual.reliability;
strKr.Local := inLocal.value AND inLocal.reliability;
strKr.Distance := inDistance.value AND inDistance.reliability;
strKr.ErrorPowerOff := inErrorPowerOff.value AND inErrorPowerOff.reliability;
strKr.ErrorBlock := inErrorBlock.value AND inErrorBlock.reliability;
strKr.OpcCommandsDisabled := strKr.inOpcCommandsDisabled;

(* ---- Формирование признака блокировки Открытия крана по высокому давлению ---- *)
	IF strKr.ISVALIDREF_inDp THEN

		strKr.Dp := NOT inDp.value AND inDp.reliability;

		dP_Trig(CLK := strKr.Dp );
		dP_Trig_reliability(CLK :=NOT inDp.reliability);

		IF dP_Trig.Q OR dP_Trig_reliability.Q THEN
			BlockedOpenControl := TRUE;
		END_IF;
		(* ---- автоматический сброс *)
		resetBlockedOpenControl_Trig(CLK := (inDp.value) AND inDp.reliability);
		IF resetBlockedOpenControl_Trig.Q THEN
			BlockedOpenControl := FALSE;
		END_IF;
	ELSE
		strKr.Dp  := FALSE;
		BlockedOpenControl := FALSE;
	END_IF;

(* ---- Формирование признака сдвига ---- *)
getSdvig := FALSE;
IF (strKr.ISVALIDREF_cmdOn OR strKr.ISVALIDREF_cmdOff) AND NOT strKr.Local THEN
	IF NOT (strKr.CmdOn OR strKr.CmdOff) THEN
		IF (lastOnStatus <> strKr.onStatus AND
		(strKr.onStatus <> _statusDualInput.STATUS_NOTDEFINED AND strKr.onStatus <> _statusDualInput.STATUS_ERROR) AND
		(lastOnStatus <> _statusDualInput.STATUS_NOTDEFINED AND lastOnStatus <> _statusDualInput.STATUS_ERROR)) THEN
			strKr.sdvig   := TRUE;
		END_IF;
	END_IF;
END_IF;

IF getSdvig THEN strKr.sdvig:= TRUE; END_IF;

sdvigReset(IN:=strKr.sdvig, PT:=T#15S);

IF sdvigReset.Q THEN strKr.sdvig:=FALSE; END_IF;

lastOnStatus := strKr.onStatus;

(* ---- Распаковка команды ---- *)
_sunpackerCommand(command := strKr.inCommand);
	cmd := _sunpackerCommand.cmd;
	source := _sunpackerCommand.source;

(* ---- Обработка команды ---- *)
IF cmd <> 0 AND lastCmd <> cmd and (((NOT strKr.opcCommandsDisabled) AND source > 0) OR source = 0) then
	CASE BYTE_TO_INT(cmd) OF
	(*cmd_open*) 1 :
			IF NOT BlockedOpenControl THEN
                              IF  strKr.ISVALIDREF_cmdOn THEN strKr.CmdOn := TRUE;
				IF strKr.ISVALIDREF_cmdOff THEN strKr.CmdOff := FALSE; END_IF;
			ELSIF  strKr.ISVALIDREF_cmdOff THEN strKr.CmdOff := FALSE;  END_IF;
			errorCMDTimer(IN := false);

			_commandErrorTimer := true;
			strKr.lastCmdIsOn := true;
                              END_IF;
	(*cmd_close*) 2 :
			IF strKr.ISVALIDREF_cmdOff THEN strKr.CmdOff := TRUE;
				IF strKr.ISVALIDREF_cmdOn THEN strKr.CmdOn := FALSE; END_IF;
			ELSIF strKr.ISVALIDREF_cmdOn THEN strKr.CmdOn := FALSE; END_IF;
			errorCMDTimer(IN := false);

			_commandErrorTimer := true;
			strKr.lastCmdIsOn := false;
	(*cmd_reset*) 3 :   IF (strKr.ISVALIDREF_statOn) OR (strKr.ISVALIDREF_statOff) THEN
			strKr.CmdOn := FALSE;
			strKr.CmdOff := FALSE;
                              lastCmd := 0;
			_commandErrorTimer := false;
			strKr.lastCmdIsOn := false;
                              END_IF;

	END_CASE;
	source_for_Status := source;
	cmd_for_Status := cmd;
	command_error_for_Status := 0;
END_IF;
lastCmd := cmd;

errorCMDTimer(In := _commandErrorTimer, PT :=T#90s);

continueHoldCommandTimer(IN:=(strKr.onStatus = _statusDualInput.STATUS_ON) OR
(strKr.onStatus = _statusDualInput.STATUS_OFF), PT:=strKr.continueHoldCommand);

(* ---- алгоритм  для команды ВКЛючить ---- *)
IF (strKr.onStatus = _statusDualInput.STATUS_ON) and strKr.lastCmdIsOn  then
	IF strKr.ISVALIDREF_cmdOn AND strKr.ISVALIDREF_cmdOff then
          IF continueHoldCommandTimer.Q THEN
          strKr.cmdOn := false; END_IF;
          END_IF;
	 errorCMDTimer(In := false);
	 _commandErrorTimer := false;
	 cmd_for_Status := 0;
	 source_for_Status := 0;
END_IF;

(* ---- off ---- *)
IF (strKr.onStatus = _statusDualInput.STATUS_OFF) and  (NOT strKr.lastCmdIsOn) then
	IF strKr.ISVALIDREF_cmdOn AND strKr.ISVALIDREF_cmdOff then
          IF continueHoldCommandTimer.Q THEN
          strKr.cmdOff := false; END_IF;
          END_IF;
	 errorCMDTimer(In := false);
	 _commandErrorTimer := false;
	 cmd_for_Status := 0;
	 source_for_Status := 0;
END_IF;

(* ---- ошибка исполнения команды ---- *)
if errorCMDTimer.Q and (cmd_for_Status <> 0) then
	command_error_for_Status :=  cmd_for_Status;
	_commandErrorTimer := false;
	strKr.CmdOn := false;
	strKr.CmdOff := false;
	(*lastCmd := 0;*)
END_IF;

(* ---- сброс ошибки команды ---- *)
strKr.CommandFault := command_error_for_Status <> 0;
_errorReset(IN := command_error_for_Status <> 0, PT := T#5S);
IF _errorReset.Q THEN
	cmd_for_Status := 0;
	source_for_Status := 0;
	command_error_for_Status := 0;

END_IF;

outputsSets(in := (strKr.ISVALIDREF_cmdOn and strKr.cmdOn ) OR (strKr.ISVALIDREF_cmdOff and strKr.cmdOff), PT := T#2S);
	IF NOT outputsSets.Q THEN
		strKr.So := inSo._inversed AND inSo.reliability AND strKr.ISVALIDREF_inSo;
		strKr.Sz := inSz._inversed AND inSz.reliability AND strKr.ISVALIDREF_inSz;
	END_IF;

cmdOn := strKr.cmdOn;
cmdOff:= strKr.cmdOff;

(* ---- формирование зашифрованного статуса для АРМа ---- *)
strKr.status := shl(BYTE_TO_DWORD(source_for_Status), 29)
		OR shl(BYTE_TO_DWORD(cmd_for_Status), 26)
		OR shl(BYTE_TO_DWORD(command_error_for_Status), 23)
		OR shl(bool_to_DWORD(strKr.sdvig), 22)
		OR shl(bool_to_DWORD(strKr.OpcCommandsDisabled), 21)
                    OR shl(bool_to_DWORD(strKr.Dp), 14)
                    OR shl(BOOL_TO_DWORD(strKr.Sz), 13)
		OR shl(BOOL_TO_DWORD(strKr.So), 12)
		OR shl(BOOL_TO_DWORD(strKr.ErrorBlock), 11)
		OR shl(BOOL_TO_DWORD(strKr.ErrorPowerOff), 10)
		OR shl(BOOL_TO_DWORD(strKr.Manual), 8)
		OR shl(BOOL_TO_DWORD(strKr.Auto), 7)
		OR shl(BOOL_TO_DWORD(strKr.Distance), 6)
		OR shl(BOOL_TO_DWORD(strKr.Local), 5)
		OR shl(BOOL_TO_DWORD(strKr.Ns), 4)
                	OR shl(BOOL_TO_DWORD(strKr.Accident ),3)
		OR BYTE_TO_DWORD(strKr.onStatus);

(* ---- fb_Kran_Init.st ---- *)
FUNCTION_BLOCK fb_Kran_Init

VAR_INPUT
	data_Ini : BOOL; (*Флаг необходимости инициализации параметров.*)
	ISVALIDREF_statOn : BOOL;
	ISVALIDREF_statOff : BOOL;
	ISVALIDREF_cmdOn : BOOL;
	ISVALIDREF_cmdOff : BOOL;
	ISVALIDREF_inSo : BOOL;
	ISVALIDREF_inSz : BOOL;
	ISVALIDREF_inDp : BOOL          := False;
	continueHoldCommand : TIME;
END_VAR

VAR_IN_OUT
	str_Kr : struct_Kran; (*Дескриптор AI-канала.*)
END_VAR

VAR_OUTPUT
	Init : BOOL          := FALSE; (*Флаг успешно выполненной инициализации.*)
END_VAR

(*****            Функциональный блок переинициализации структуры  Kran          *****)

        Init := False;

    IF data_Ini THEN                            (* Параметрам требуется переинициализация. *)
        str_Kr.ISVALIDREF_statOn                := ISVALIDREF_statOn;
        str_Kr.ISVALIDREF_statOff               := ISVALIDREF_statOff;
        str_Kr.ISVALIDREF_cmdOn                 := ISVALIDREF_cmdOn;
        str_Kr.ISVALIDREF_cmdOff                := ISVALIDREF_cmdOff;
        str_Kr.ISVALIDREF_inSo                  := ISVALIDREF_inSo;
        str_Kr.ISVALIDREF_inSz                  := ISVALIDREF_inSz;
        str_Kr.ISVALIDREF_inDp                  := ISVALIDREF_inDp;
        str_Kr.continueHoldCommand              := continueHoldCommand;

        data_Ini:=False;
        Init := TRUE;
   END_IF;
 IF Init THEN
        ISVALIDREF_statOn:= false;
        ISVALIDREF_statOff:= false;
        ISVALIDREF_cmdOn:= false;
        ISVALIDREF_cmdOff:= false;
        ISVALIDREF_inSo:= false;
        ISVALIDREF_inSz:= false;
        ISVALIDREF_inDp:= false;
        continueHoldCommand:= T#0S;
  END_IF;

(* ---- fb_KranOpenProtection.st ---- *)
FUNCTION_BLOCK fb_KranOpenProtection

VAR_INPUT
	im : struct_Kran;
END_VAR

VAR_IN_OUT
	StrDIp : struct_DiProtection;
END_VAR

VAR
	_sunpackerCommand : fb_sunpackerCommand;
	statusDualInput : TYPE_statusDualInput;
	_ProtectionTags : TYPE_ProtectionTags;
	_signalingTp : TOF;
	timer : TON;
	SignalingTrig : R_TRIG;
	SignalingFTrig : F_TRIG;
	SignalingDi : BOOL;
	source : BYTE;
	cmd : BYTE;
	lastCmd : BYTE;
	source_for_Status : BYTE;
	cmd_for_Status : BYTE;
	command_error_for_Status : BYTE;
	resetCmdTimer : TON;
	resetCmdTimerPriznak : BOOL;
	signalinTimer : TON;
	runOnStart_Trig : R_TRIG;
END_VAR

timer(IN := (im.onStatus<>statusDualInput.STATUS_ON) AND StrDIp.isRunning  , PT := StrDIp.delay);
SignalingTrig(CLK := timer.Q);
IF SignalingTrig.Q THEN
	SignalingDi := TRUE;
END_IF;
SignalingFTrig(CLK := timer.Q);
IF SignalingFTrig.Q THEN
	SignalingDi := FALSE;
END_IF;

StrDIp.Tag := StrDIp.inTag;
StrDIp.RunOnStart := StrDIp.inRunOnStart;

StrDIp.CanRun := StrDIp.inCanRun;

StrDIp.OpcCommandsDisabled := StrDIp.inOpcCommandsDisabled;

(* ---- Если управление с ВУ заблокировано, то передаем команду из алгоритма ---- *)
IF StrDIp.inOpcCommandsDisabled THEN
	StrDIp.inCommand := StrDIp.inCommand_Alg;
ELSE (* иначе передаем команду с АРМа*)
	StrDIp.inCommand := StrDIp.inCommand_ARM;
END_IF;

_sunpackerCommand(command := StrDIp.inCommand);
	source := _sunpackerCommand.source;
	cmd := _sunpackerCommand.cmd;

IF cmd <> 0 AND lastCmd <> cmd AND (((NOT StrDIp.opcCommandsDisabled) AND source > 0) OR source = 0) then
	CASE BYTE_TO_INT(cmd) OF
	        (*cmdRun*) 1: 	IF        NOT StrDIp.Remont THEN
					StrDIp.isEnded := FALSE;
					StrDIp.hasError 	:= FALSE;
					StrDIp.isRunning := TRUE;
					cmd_for_Status := cmd;
					source_for_Status := source;
					command_error_for_Status := 0;
				ELSE
					StrDIp.isRunning := FALSE;
					StrDIp.isEnded := FALSE;
					StrDIp.hasError 	:= FALSE;

					cmd_for_Status := 0;
					source_for_Status := source;
					command_error_for_Status := cmd;
				END_IF;
                                        StrDIp.inOpcCommandsDisabled:=FALSE;

                (*cmdReset*) 2: 	StrDIp.isRunning := FALSE;
				StrDIp.isEnded := FALSE;
				StrDIp.hasError 	:= FALSE;
				SignalingDi:= FALSE;
				StrDIp.Check := FALSE;
				cmd_for_Status := cmd;
				source_for_Status := source;
				command_error_for_Status := 0;
                                        StrDIp.inOpcCommandsDisabled:=FALSE;

	(*cmd_setRemont*) 4 :	StrDIp.Remont := TRUE;
				(*StrDIp.isRunning := FALSE;*)

				cmd_for_Status := cmd;
				source_for_Status := source;
				command_error_for_Status := 0;

        (*cmd_resetRemont*) 5 : 	(*IF (im.onStatus<>statusDualInput.STATUS_ON) THEN
					cmd_for_Status := 0;
					source_for_Status := 0;
					command_error_for_Status := cmd;
				ELSE*)
					StrDIp.Remont := FALSE;
					(*StrDIp.isRunning := TRUE;*)

					cmd_for_Status := cmd;
					source_for_Status := source;
					command_error_for_Status := 0;
				(*END_IF;*)

	(*cmd_setCheck*) 6 : 	StrDIp.Check := TRUE;

				cmd_for_Status := cmd;
				source_for_Status := source;
				command_error_for_Status := 0;
	END_CASE;
	resetCmdTimer(IN := false);
	resetCmdTimerPriznak := TRUE;
END_IF;
lastCmd := cmd;

resetCmdTimer(IN := resetCmdTimerPriznak);
IF resetCmdTimer.Q THEN
	resetCmdTimerPriznak := FALSE;
	source_for_Status := 0;
	cmd_for_Status := 0;
	command_error_for_Status := 0;
END_IF;

IF StrDIp.isRunning AND  NOT StrDIp.Remont AND NOT StrDIp.Check THEN
	StrDIp.Signaling := SignalingDi;
	StrDIp.SignalingTP := _signalingTp.Q;
ELSE
	StrDIp.Signaling := 0;
	StrDIp.SignalingTP := 0;
END_IF;

_signalingTp(in := StrDIp.Signaling, PT := T#1s);

StrDIp.status :=  SHL(BYTE_TO_DWORD(source_for_Status), 29)
			OR SHL(BYTE_TO_DWORD(cmd_for_Status), 26)
			OR SHL(BYTE_TO_DWORD(command_error_for_Status), 23)
			OR SHL(BOOL_TO_DWORD(StrDIp.OpcCommandsDisabled ), 21)
			OR SHL(BOOL_TO_DWORD(StrDIp.Signaling), 16)
			OR SHL(BOOL_TO_DWORD(StrDIp.RunOnStart ), 15)
			OR SHL(BOOL_TO_DWORD(StrDIp.remont), 6)
			OR SHL(BOOL_TO_DWORD(StrDIp.Check), 5)
			OR SHL(BOOL_TO_DWORD(StrDIp.hasError), 4)
			OR SHL(BOOL_TO_DWORD(StrDIp.SignalingTP), 3)
			OR SHL(BOOL_TO_DWORD(StrDIp.CanRun), 2)
			OR SHL(BOOL_TO_DWORD(StrDIp.isEnded), 1)
			OR BOOL_TO_DWORD(StrDIp.isRunning);

(* ---- fb_meandr.st ---- *)
FUNCTION_BLOCK fb_meandr

VAR
	_output : BOOL;
END_VAR

VAR_INPUT
	period : TIME          := T#300MS;
END_VAR

VAR
	timer : TON;
	FALSE_val : BOOL          := FALSE;
	TRUE_val : BOOL          := TRUE;
END_VAR

VAR_IN_OUT
	output : BOOL;
END_VAR

timer(in:=NOT FALSE_val,PT:=period);

IF timer.Q THEN
    _output:=_output XOR TRUE_val;
    timer(in:=FALSE);
END_IF;

output:=_output;

(* ---- fb_MvProtection.st ---- *)
FUNCTION_BLOCK fb_MvProtection

VAR_INPUT
	sw : struct_SectionSwitch;
END_VAR

VAR_IN_OUT
	StrDIp : struct_DiProtection;
END_VAR

VAR
	_sunpackerCommand : fb_sunpackerCommand;
	statusDualInput : TYPE_statusDualInput;
	_ProtectionTags : TYPE_ProtectionTags;
	_signalingTp : TOF;
	timer : TON;
	SignalingTrig : R_TRIG;
	SignalingFTrig : F_TRIG;
	SignalingDi : BOOL;
	source : BYTE;
	cmd : BYTE;
	lastCmd : BYTE;
	source_for_Status : BYTE;
	cmd_for_Status : BYTE;
	command_error_for_Status : BYTE;
	resetCmdTimer : TON;
	resetCmdTimerPriznak : BOOL;
	signalinTimer : TON;
	runOnStart_Trig : R_TRIG;
END_VAR

timer(IN := (sw.onStatus = statusDualInput.STATUS_OFF) AND StrDIp.isRunning  , PT := StrDIp.delay);
SignalingTrig(CLK := timer.Q);
IF SignalingTrig.Q THEN
	SignalingDi := TRUE;
END_IF;
SignalingFTrig(CLK := timer.Q);
IF SignalingFTrig.Q THEN
	SignalingDi := FALSE;
END_IF;

StrDIp.Tag := StrDIp.inTag;
StrDIp.RunOnStart := StrDIp.inRunOnStart;

StrDIp.CanRun := StrDIp.inCanRun;

StrDIp.OpcCommandsDisabled := StrDIp.inOpcCommandsDisabled;

(* ---- Если управление с ВУ заблокировано, то передаем команду из алгоритма ---- *)
IF StrDIp.inOpcCommandsDisabled THEN
	StrDIp.inCommand := StrDIp.inCommand_Alg;
ELSE (* иначе передаем команду с АРМа*)
	StrDIp.inCommand := StrDIp.inCommand_ARM;
END_IF;

_sunpackerCommand(command := StrDIp.inCommand);
	source := _sunpackerCommand.source;
	cmd := _sunpackerCommand.cmd;

IF cmd <> 0 AND lastCmd <> cmd AND (((NOT StrDIp.opcCommandsDisabled) AND source > 0) OR source = 0) then
	CASE BYTE_TO_INT(cmd) OF
	        (*cmdRun*) 1: 	IF        NOT StrDIp.Remont THEN
					StrDIp.isEnded := FALSE;
					StrDIp.hasError 	:= FALSE;
					StrDIp.isRunning := TRUE;
					cmd_for_Status := cmd;
					source_for_Status := source;
					command_error_for_Status := 0;
				ELSE
					StrDIp.isRunning := FALSE;
					StrDIp.isEnded := FALSE;
					StrDIp.hasError 	:= FALSE;

					cmd_for_Status := 0;
					source_for_Status := source;
					command_error_for_Status := cmd;
				END_IF;
                                        StrDIp.inOpcCommandsDisabled:=FALSE;

                (*cmdReset*) 2: 	StrDIp.isRunning := FALSE;
				StrDIp.isEnded := FALSE;
				StrDIp.hasError 	:= FALSE;
				SignalingDi:= FALSE;
				StrDIp.Check := FALSE;
				cmd_for_Status := cmd;
				source_for_Status := source;
				command_error_for_Status := 0;
                                        StrDIp.inOpcCommandsDisabled:=FALSE;

	(*cmd_setRemont*) 4 :	StrDIp.Remont := TRUE;
				(*StrDIp.isRunning := FALSE;*)

				cmd_for_Status := cmd;
				source_for_Status := source;
				command_error_for_Status := 0;

        (*cmd_resetRemont*) 5 : 	(*IF (sw.onStatus = statusDualInput.STATUS_OFF) THEN
					cmd_for_Status := 0;
					source_for_Status := 0;
					command_error_for_Status := cmd;
				ELSE*)
					StrDIp.Remont := FALSE;
					(*StrDIp.isRunning := TRUE;*)

					cmd_for_Status := cmd;
					source_for_Status := source;
					command_error_for_Status := 0;
				(*END_IF;*)

	(*cmd_setCheck*) 6 : 	StrDIp.Check := TRUE;

				cmd_for_Status := cmd;
				source_for_Status := source;
				command_error_for_Status := 0;
	END_CASE;
	resetCmdTimer(IN := false);
	resetCmdTimerPriznak := TRUE;
END_IF;
lastCmd := cmd;

resetCmdTimer(IN := resetCmdTimerPriznak);
IF resetCmdTimer.Q THEN
	resetCmdTimerPriznak := FALSE;
	source_for_Status := 0;
	cmd_for_Status := 0;
	command_error_for_Status := 0;
END_IF;

IF StrDIp.isRunning AND  NOT StrDIp.Remont AND NOT StrDIp.Check THEN
	StrDIp.Signaling := SignalingDi;
	StrDIp.SignalingTP := _signalingTp.Q;
ELSE
	StrDIp.Signaling := 0;
	StrDIp.SignalingTP := 0;
END_IF;

_signalingTp(in := StrDIp.Signaling, PT := T#1s);

StrDIp.status :=  SHL(BYTE_TO_DWORD(source_for_Status), 29)
			OR SHL(BYTE_TO_DWORD(cmd_for_Status), 26)
			OR SHL(BYTE_TO_DWORD(command_error_for_Status), 23)
			OR SHL(BOOL_TO_DWORD(StrDIp.OpcCommandsDisabled ), 21)
			OR SHL(BOOL_TO_DWORD(StrDIp.Signaling), 16)
			OR SHL(BOOL_TO_DWORD(StrDIp.RunOnStart ), 15)
			OR SHL(BOOL_TO_DWORD(StrDIp.remont), 6)
			OR SHL(BOOL_TO_DWORD(StrDIp.Check), 5)
			OR SHL(BOOL_TO_DWORD(StrDIp.hasError), 4)
			OR SHL(BOOL_TO_DWORD(StrDIp.SignalingTP), 3)
			OR SHL(BOOL_TO_DWORD(StrDIp.CanRun), 2)
			OR SHL(BOOL_TO_DWORD(StrDIp.isEnded), 1)
			OR BOOL_TO_DWORD(StrDIp.isRunning);

(* ---- fb_OilPump.st ---- *)
FUNCTION_BLOCK fb_OilPump

VAR_INPUT
	statOn : BOOL;
	statOff : BOOL;
	statOn_reliability : BOOL;
	statOff_reliability : BOOL;
END_VAR

VAR_IN_OUT
	StrSw : struct_OilPump;
END_VAR

VAR_INPUT
	inNs : TYPE_ReliableBit;
	inAccident : TYPE_ReliableBit;
	inLocal : TYPE_ReliableBit;
	inDistance : TYPE_ReliableBit;
	inBreakCmdOn : TYPE_ReliableBit;
	inBreakCmdOff : TYPE_ReliableBit;
END_VAR

VAR
	onInit : BOOL          := FALSE;
	_statOn : BOOL;
	_statOff : BOOL;
	getSdvig : BOOL;
	lastOnStatus : BYTE;
	cmd : BYTE;
	source : BYTE;
	lastCmd : BYTE;
	source_for_Status : BYTE;
	cmd_for_Status : BYTE;
	command_error_for_Status : BYTE;
	_sunpackerCommand : fb_sunpackerCommand;
	_statusDualInput : TYPE_statusDualInput;
	_commandDualInput : TYPE_commandDualInput;
	_commandErrorTimer : BOOL;
	resetErrorTimer : BOOL;
	_changWithoutCommand : BOOL;
	errorCMDTimer : TON;
	sdvigReset : TON;
	_errorReset : TON;
	outputsSets : TOF;
END_VAR

VAR_IN_OUT
	cmdOn : BOOL;
	cmdOff : BOOL;
END_VAR

IF NOT onInit THEN
IF StrSw.ISVALIDREF_cmdOn XOR StrSw.ISVALIDREF_cmdOff THEN
	IF 	StrSw.ISVALIDREF_cmdOn THEN
		lastCmd:= 2; (*baseCmdOff*)
	ELSE
		lastCmd:= 1; (*baseCmdOn*)
	END_IF;
END_IF;
onInit:=TRUE;
END_IF;

(* ---- Если управление с ВУ заблокировано, то в ИМ передаем команду из алгоритма ---- *)
IF StrSw.inOpcCommandsDisabled THEN
	StrSw.inCommand := StrSw.inCommand_Alg;
ELSE (* иначе передаем команду с АРМа*)
	StrSw.inCommand := StrSw.inCommand_ARM;
END_IF;

(* ---- Формирование состояния механизма ---- *)

IF (StrSw.ISVALIDREF_statOn) OR (StrSw.ISVALIDREF_statOff) THEN
	IF (StrSw.ISVALIDREF_statOn) AND (StrSw.ISVALIDREF_statOff) THEN
	StrSw.reliability:= statOn_reliability AND statOff_reliability;
		_statOn  := statOn;
		_statOff := statOff;
	ELSIF (StrSw.ISVALIDREF_statOn) THEN
                     StrSw.reliability:= statOn_reliability;
		_statOn  := statOn;
		_statOff := NOT statOn;
	ELSIF (StrSw.ISVALIDREF_statOff) THEN
		 StrSw.reliability:= statOff_reliability;
		_statOn  := NOT statOff;
		_statOff :=statOff;
	END_IF;

	IF StrSw.reliability THEN
		IF _statOn AND NOT _statOff 		THEN 	StrSw.onStatus := _statusDualInput.STATUS_ON;
		ELSIF _statOff AND NOT _statOn 	THEN 	StrSw.onStatus := _statusDualInput.Status_OFF;
		ELSIF NOT _statOn AND NOT _statOff 	THEN 	StrSw.onStatus := _statusDualInput.STATUS_TRANSITIONAL;
		ELSE					StrSw.onStatus := _statusDualInput.STATUS_ERROR;
                    END_IF;

	ELSE
		StrSw.onStatus := _statusDualInput.STATUS_NOTDEFINED;

	END_IF;
ELSE
	CASE BYTE_TO_INT(lastCmd) OF
		(*baseCmdOn*) 1: StrSw.onStatus  := _statusDualInput.STATUS_ON;
		(*baseCmdOff*) 2: StrSw.onStatus  := _statusDualInput.STATUS_OFF;

	ELSE
		 StrSw.onStatus := _statusDualInput.STATUS_NOTDEFINED;

	END_CASE;
END_IF;

StrSw.Accident := inAccident.value AND inAccident.reliability;
StrSw.Ns := inNs.value AND inNs.reliability;
StrSw.Local := inLocal.value AND inLocal.reliability;
StrSw.Distance := inDistance.value AND inDistance.reliability;
StrSw.OpcCommandsDisabled := StrSw.inOpcCommandsDisabled;

StrSw.Blocked:=StrSw.Accident OR StrSw.Local OR StrSw.breakCmdOn OR StrSw.breakCmdOff OR StrSw.inBlocked;

StrSw.Rezervny:=NOT StrSw.Osnovnoy;

(* ---- Формирование признака сдвига ---- *)

getSdvig := FALSE;
IF (StrSw.ISVALIDREF_cmdOn OR StrSw.ISVALIDREF_cmdOff) AND NOT StrSw.Local THEN
	IF NOT (StrSw.CmdOn OR StrSw.CmdOff) THEN
                     IF (lastOnStatus <> StrSw.onStatus AND
		(StrSw.onStatus <> _statusDualInput.STATUS_NOTDEFINED AND
                     StrSw.onStatus <> _statusDualInput.STATUS_ERROR)     AND
		(lastOnStatus <> _statusDualInput.STATUS_NOTDEFINED   AND
                     lastOnStatus <> _statusDualInput.STATUS_ERROR))
                    THEN
			getSdvig   := TRUE;
		END_IF;
	END_IF;
END_IF;

IF getSdvig THEN StrSw.sdvig:= TRUE; END_IF;

sdvigReset(IN:=StrSw.sdvig, PT:=T#15S);

IF sdvigReset.Q THEN StrSw.sdvig:=FALSE; END_IF;

lastOnStatus := StrSw.onStatus;

(* ---- Распаковка команды ---- *)
_sunpackerCommand(command := StrSw.inCommand);
	cmd := _sunpackerCommand.cmd;
	source := _sunpackerCommand.source;

(* ---- Обработка команды ---- *)
IF cmd <> 0 AND lastCmd <> cmd and (((NOT StrSw.opcCommandsDisabled) AND source > 0) OR source = 0) then
	CASE BYTE_TO_INT(cmd) OF
	(*cmd_on*) 1 :
			IF  StrSw.ISVALIDREF_cmdOn THEN StrSw.CmdOn := TRUE;
				IF StrSw.ISVALIDREF_cmdOff THEN StrSw.CmdOff := FALSE; END_IF;
			ELSIF  StrSw.ISVALIDREF_cmdOff THEN StrSw.CmdOff := FALSE;  END_IF;
			errorCMDTimer(IN := false);
			_commandErrorTimer := true;
			StrSw.lastCmdIsOn := true;
	(*cmd_off*) 2 :
			IF StrSw.ISVALIDREF_cmdOff THEN StrSw.CmdOff := TRUE;
				IF StrSw.ISVALIDREF_cmdOn THEN StrSw.CmdOn := FALSE; END_IF;
			ELSIF StrSw.ISVALIDREF_cmdOn THEN StrSw.CmdOn := FALSE; END_IF;
			errorCMDTimer(IN := false);

			_commandErrorTimer := true;
			StrSw.lastCmdIsOn := false;
	(*cmd_reset*) 3 :    IF StrSw.ISVALIDREF_statOn OR StrSw.ISVALIDREF_statOff THEN
			StrSw.CmdOn := FALSE;
			StrSw.CmdOff := FALSE;
                              lastCmd := 0;
			_commandErrorTimer := false;
			StrSw.lastCmdIsOn := false;
                               END_IF;
	END_CASE;
	source_for_Status := source;
	cmd_for_Status := cmd;
	command_error_for_Status := 0;
END_IF;

lastCmd := cmd;
errorCMDTimer(In := _commandErrorTimer, PT :=T#10s);

(* ---- алгоритм  для команды ВКЛючить ---- *)
IF (StrSw.onStatus = _statusDualInput.STATUS_ON) and StrSw.lastCmdIsOn then
	IF StrSw.ISVALIDREF_cmdOn AND StrSw.ISVALIDREF_cmdOff then  StrSw.cmdOn := false; END_IF;

	 errorCMDTimer(In := false);
	 _commandErrorTimer := false;
	 cmd_for_Status := 0;
	 source_for_Status := 0;
END_IF;

(* ---- off ---- *)
IF (StrSw.onStatus = _statusDualInput.STATUS_OFF) and (NOT StrSw.lastCmdIsOn) then
	IF StrSw.ISVALIDREF_cmdOn AND StrSw.ISVALIDREF_cmdOff then  StrSw.cmdOff := false; END_IF;

	 errorCMDTimer(In := false);
	 _commandErrorTimer := false;
	 cmd_for_Status := 0;
	 source_for_Status := 0;
END_IF;

(* ---- ошибка исполнения команды ---- *)
if errorCMDTimer.Q and (cmd_for_Status <> 0) then
	command_error_for_Status :=  cmd_for_Status;
	_commandErrorTimer := false;
	StrSw.CmdOn := false;
	StrSw.CmdOff := false;
	lastCmd := 0;
end_if;

(* ---- сброс ошибки команды ---- *)
StrSw.CommandFault := command_error_for_Status <> 0;
_errorReset(IN := command_error_for_Status <> 0, PT := T#5S);
IF _errorReset.Q THEN
	cmd_for_Status := 0;
	source_for_Status := 0;
	command_error_for_Status := 0;
END_IF;

outputsSets(in := (StrSw.ISVALIDREF_cmdOn and StrSw.cmdOn ) OR (StrSw.ISVALIDREF_cmdOff and StrSw.cmdOff), PT := T#2S);
	IF NOT outputsSets.Q THEN
		StrSw.BreakCmdOn := inBreakCmdOn._inversed AND inBreakCmdOn.reliability AND StrSw.ISVALIDREF_inBreakCmdOn;
		StrSw.BreakCmdOff := inBreakCmdOff._inversed AND inBreakCmdOff.reliability AND StrSw.ISVALIDREF_inBreakCmdOff;
	END_IF;

cmdOn := StrSw.cmdOn;
cmdOff:= StrSw.cmdOff;

(* ---- формирование зашифрованного статуса для АРМа ---- *)
StrSw.status := shl(BYTE_TO_DWORD(source_for_Status), 29)
		OR shl(BYTE_TO_DWORD(cmd_for_Status), 26)
		OR shl(BYTE_TO_DWORD(command_error_for_Status), 23)
		OR shl(bool_to_DWORD(StrSw.sdvig), 22)
		OR shl(bool_to_DWORD(StrSw.OpcCommandsDisabled), 21)
                    OR shl(bool_to_DWORD(StrSw.lastCmdIsOn), 14)
                    OR shl(BOOL_TO_DWORD(StrSw.BreakCmdOff), 13)
		OR shl(BOOL_TO_DWORD(StrSw.BreakCmdOn), 12)
		OR shl(BOOL_TO_DWORD(StrSw.Distance), 6)
		OR shl(BOOL_TO_DWORD(StrSw.Local), 5)
		OR shl(BOOL_TO_DWORD(StrSw.Ns), 4)
                	OR shl(BOOL_TO_DWORD(StrSw.Accident ),3)
		OR BYTE_TO_DWORD(StrSw.onStatus);

(* ---- fb_OilPump_Init.st ---- *)
FUNCTION_BLOCK fb_OilPump_Init

VAR_INPUT
	data_Ini : BOOL; (*Флаг необходимости инициализации параметров.*)
	ISVALIDREF_statOn : BOOL;
	ISVALIDREF_statOff : BOOL;
	ISVALIDREF_cmdOn : BOOL;
	ISVALIDREF_cmdOff : BOOL;
	ISVALIDREF_inBreakCmdOn : BOOL;
	ISVALIDREF_inBreakCmdOff : BOOL;
END_VAR

VAR_IN_OUT
	str_Op : struct_OilPump;
END_VAR

VAR_OUTPUT
	Init : BOOL          := FALSE; (*Флаг успешно выполненной инициализации.*)
END_VAR

(*****            Функциональный блок переинициализации структуры  НУ          *****)

 Init := FALSE;

    IF data_Ini THEN                            (* Параметрам требуется переинициализация. *)
        str_Op.ISVALIDREF_statOn                := ISVALIDREF_statOn;
        str_Op.ISVALIDREF_statOff               := ISVALIDREF_statOff;
        str_Op.ISVALIDREF_cmdOn                 := ISVALIDREF_cmdOn;
        str_Op.ISVALIDREF_cmdOff                := ISVALIDREF_cmdOff;
        str_Op.ISVALIDREF_inBreakCmdOn          := ISVALIDREF_inBreakCmdOn;
        str_Op.ISVALIDREF_inBreakCmdOff         := ISVALIDREF_inBreakCmdOff;
        data_Ini:=FALSE;
        Init := TRUE;
    END_IF;

        ISVALIDREF_statOn:= FALSE;
        ISVALIDREF_statOff:= FALSE;
        ISVALIDREF_cmdOn:= FALSE;
        ISVALIDREF_cmdOff:= FALSE;
        ISVALIDREF_inBreakCmdOn:= FALSE;
        ISVALIDREF_inBreakCmdOff:= FALSE;

(* ---- fb_ph_AIprotection.st ---- *)
FUNCTION_BLOCK fb_ph_AIprotection

VAR_IN_OUT
	StrAiP : struct_AiProtection;
END_VAR

VAR_INPUT
	act : TYPE_PhaseAlgoritmAction;
	PhaseNumber : UINT;
END_VAR

VAR_IN_OUT
	StrPh : struct_PhaseAlgoritm;
END_VAR

VAR
	CommandFault_Trig : R_TRIG;
	reset_Trig : R_TRIG;
	_statusDualInput : TYPE_statusDualInput;
END_VAR

IF StrPh.run AND NOT StrPh.start THEN
	StrPh.start := TRUE;
	StrPh.top := FALSE;
	StrPh.error := FALSE;
          StrPh.run:=FALSE;

	CASE act OF
		(*PhaseAlgoritmAction.run*)    _run : runAiProtection(StrAiP); (*cmd_run*)
		(*PhaseAlgoritmAction.reset*)_reset : resetAiProtection(StrAiP); (*cmd_reset*)
	END_CASE;
END_IF;

IF StrPh.start AND NOT StrPh.top THEN
                    CommandFault_Trig(CLK := StrAiP.hasError);
                    IF CommandFault_Trig.Q THEN
	          StrPh.error := TRUE;
                    END_IF;

		CASE act OF
		(*PhaseAlgoritmAction.run*)    _run:    StrPh.top:=StrAiP.isRunning;

		(*PhaseAlgoritmAction.reset*) _reset:   StrPh.top := NOT StrAiP.isRunning;
		END_CASE;

END_IF;

IF StrPh.top THEN
StrPh.error := FALSE;
END_IF;

reset_Trig(CLK := StrPh.reset);
IF reset_Trig.Q THEN
          StrPh.start := FALSE;
	StrPh.error := FALSE;
	StrPh.top := FALSE;
          StrPh.run:=FALSE;
          StrPh.reset:=FALSE;
END_IF;

StrPh.startStatus := SHL(BOOL_TO_DWORD(StrPh.start), PhaseNumber);
StrPh.errorStatus := SHL(BOOL_TO_DWORD(StrPh.error), PhaseNumber);
StrPh.topStatus := SHL(BOOL_TO_DWORD(StrPh.top), PhaseNumber);

(* ---- fb_ph_algoritm.st ---- *)
FUNCTION_BLOCK fb_ph_algoritm

VAR_IN_OUT
	alg : struct_Alg;
END_VAR

VAR_INPUT
	act : TYPE_PhaseAlgoritmAction;
	PhaseNumber : UINT;
	waitCompletion : BOOL;
END_VAR

VAR_IN_OUT
	StrPh : struct_PhaseAlgoritm;
END_VAR

VAR
	CommandFault_Trig : R_TRIG;
	reset_Trig : R_TRIG;
	_statusDualInput : TYPE_statusDualInput;
END_VAR

IF StrPh.run AND NOT StrPh.start THEN
	StrPh.start := TRUE;
	StrPh.top := FALSE;
	StrPh.error := FALSE;
          StrPh.run:=FALSE;

	CASE act OF
		(*PhaseAlgoritmAction.run*)    _run : runIfNotRunning(alg); (*cmd_run*)
		(*PhaseAlgoritmAction.reset*)_reset : resetIfRunning(alg); (*cmd_reset*)
	END_CASE;
END_IF;

IF StrPh.start AND NOT StrPh.top THEN
                    CommandFault_Trig(CLK := alg.hasError);
                    IF CommandFault_Trig.Q THEN
	          StrPh.error := TRUE;
                    END_IF;

		CASE act OF
		(*PhaseAlgoritmAction.run*)    _run:
                                                        IF waitCompletion THEN
		                                	StrPh.top:=alg.isEnded;
		                                    ELSE
			                              StrPh.top:=alg.isRuning;
		                                    END_IF;

		(*PhaseAlgoritmAction.reset*) _reset:   StrPh.top := NOT alg.isRuning;
		END_CASE;

END_IF;

IF StrPh.top THEN
StrPh.error := FALSE;
END_IF;

reset_Trig(CLK := StrPh.reset);
IF reset_Trig.Q THEN
          IF waitCompletion THEN
          resetIfRunning(alg);
          END_IF;
	StrPh.start := FALSE;
	StrPh.error := FALSE;
	StrPh.top := FALSE;
          StrPh.run:=FALSE;
          StrPh.reset:=FALSE;
END_IF;

StrPh.startStatus := SHL(BOOL_TO_DWORD(StrPh.start), PhaseNumber);
StrPh.errorStatus := SHL(BOOL_TO_DWORD(StrPh.error), PhaseNumber);
StrPh.topStatus := SHL(BOOL_TO_DWORD(StrPh.top), PhaseNumber);

(* ---- fb_ph_CustomPhase.st ---- *)
FUNCTION_BLOCK fb_ph_CustomPhase

VAR_INPUT
	PhaseNumber : UINT;
END_VAR

VAR_IN_OUT
	StrPh : struct_PhaseAlgoritm;
END_VAR

VAR
	CommandFault_Trig : R_TRIG;
	reset_Trig : R_TRIG;
	_statusDualInput : TYPE_statusDualInput;
END_VAR

IF StrPh.run AND NOT StrPh.start THEN
	StrPh.start := TRUE;
	StrPh.top := FALSE;
	StrPh.error := FALSE;
          StrPh.run:=FALSE;
END_IF;

IF StrPh.top THEN StrPh.error := FALSE; END_IF;

reset_Trig(CLK := StrPh.reset);
IF reset_Trig.Q THEN
	StrPh.start := FALSE;
	StrPh.error := FALSE;
	StrPh.top := FALSE;
          StrPh.run:=FALSE;
          StrPh.reset:=FALSE;
END_IF;

StrPh.startStatus := SHL(BOOL_TO_DWORD(StrPh.start), PhaseNumber);
StrPh.errorStatus := SHL(BOOL_TO_DWORD(StrPh.error), PhaseNumber);
StrPh.topStatus := SHL(BOOL_TO_DWORD(StrPh.top), PhaseNumber);

(* ---- fb_ph_DIprotection.st ---- *)
FUNCTION_BLOCK fb_ph_DIprotection

VAR_IN_OUT
	StrDiP : struct_DiProtection;
END_VAR

VAR_INPUT
	act : TYPE_PhaseAlgoritmAction;
	PhaseNumber : UINT;
END_VAR

VAR_IN_OUT
	StrPh : struct_PhaseAlgoritm;
END_VAR

VAR
	CommandFault_Trig : R_TRIG;
	reset_Trig : R_TRIG;
	_statusDualInput : TYPE_statusDualInput;
END_VAR

IF StrPh.run AND NOT StrPh.start THEN
	StrPh.start := TRUE;
	StrPh.top := FALSE;
	StrPh.error := FALSE;
          StrPh.run:=FALSE;

	CASE act OF
		(*PhaseAlgoritmAction.run*)    _run : runDiProtection(StrDiP); (*cmd_run*)
		(*PhaseAlgoritmAction.reset*)_reset : resetDiProtection(StrDiP); (*cmd_reset*)
	END_CASE;
END_IF;

IF StrPh.start AND NOT StrPh.top THEN
                    CommandFault_Trig(CLK := StrDiP.hasError);
                    IF CommandFault_Trig.Q THEN
	          StrPh.error := TRUE;
                    END_IF;

		CASE act OF
		(*PhaseAlgoritmAction.run*)    _run:    StrPh.top:=StrDiP.isRunning;

		(*PhaseAlgoritmAction.reset*) _reset:   StrPh.top := NOT StrDiP.isRunning;
		END_CASE;

END_IF;

IF StrPh.top THEN
StrPh.error := FALSE;
END_IF;

reset_Trig(CLK := StrPh.reset);
IF reset_Trig.Q THEN
          StrPh.start := FALSE;
	StrPh.error := FALSE;
	StrPh.top := FALSE;
          StrPh.run:=FALSE;
          StrPh.reset:=FALSE;
END_IF;

StrPh.startStatus := SHL(BOOL_TO_DWORD(StrPh.start), PhaseNumber);
StrPh.errorStatus := SHL(BOOL_TO_DWORD(StrPh.error), PhaseNumber);
StrPh.topStatus := SHL(BOOL_TO_DWORD(StrPh.top), PhaseNumber);

(* ---- fb_ph_Kran.st ---- *)
FUNCTION_BLOCK fb_ph_Kran

VAR_IN_OUT
	im : struct_Kran;
	StrPh : struct_PhaseAlgoritm;
END_VAR

VAR_INPUT
	act : TYPE_DualStateImAction;
	PhaseNumber : UINT;
END_VAR

VAR
	CommandFault_Trig : R_TRIG;
	reset_Trig : R_TRIG;
	_statusDualInput : TYPE_statusDualInput;
END_VAR

IF StrPh.run AND NOT StrPh.start THEN
	StrPh.start := TRUE;
	StrPh.top := FALSE;
	StrPh.error := FALSE;
          StrPh.run:=FALSE;

	CASE act OF
		(*DualStateImAction.on*)   _on: im.inOpcCommandsDisabled:=TRUE;
                                                    im.inCommand_Alg := 1; (*cmd_open*)
		(*DualStateImAction.off*) _off: im.inOpcCommandsDisabled:=TRUE;
                                                    im.inCommand_Alg := 2; (*cmd_close*)
	END_CASE;
END_IF;

IF StrPh.start AND NOT StrPh.top THEN
                    CommandFault_Trig(CLK := im.CommandFault);
                    IF CommandFault_Trig.Q THEN
	          StrPh.error := TRUE;
                    END_IF;

		CASE act OF
		(*_DualStateImAction.on*)    _on: StrPh.top := im.onStatus = _statusDualInput.STATUS_ON;
		(*_DualStateImAction.off*)  _off: StrPh.top := im.onStatus = _statusDualInput.STATUS_OFF;
		END_CASE;

END_IF;

IF StrPh.top THEN
StrPh.error := FALSE;
END_IF;

reset_Trig(CLK := StrPh.reset);
IF reset_Trig.Q THEN
	StrPh.start := FALSE;
	StrPh.error := FALSE;
	StrPh.top := FALSE;
          StrPh.run:=FALSE;
          StrPh.reset:=FALSE;
END_IF;

StrPh.startStatus := SHL(BOOL_TO_DWORD(StrPh.start), PhaseNumber);
StrPh.errorStatus := SHL(BOOL_TO_DWORD(StrPh.error), PhaseNumber);
StrPh.topStatus := SHL(BOOL_TO_DWORD(StrPh.top), PhaseNumber);

(* ---- fb_ph_OilPump.st ---- *)
FUNCTION_BLOCK fb_ph_OilPump

VAR_IN_OUT
	im : struct_OilPump;
END_VAR

VAR_INPUT
	act : TYPE_DualStateImAction;
	PhaseNumber : UINT;
END_VAR

VAR_IN_OUT
	StrPh : struct_PhaseAlgoritm;
END_VAR

VAR
	CommandFault_Trig : R_TRIG;
	reset_Trig : R_TRIG;
	_statusDualInput : TYPE_statusDualInput;
END_VAR

IF StrPh.run AND NOT StrPh.start THEN
	StrPh.start := TRUE;
	StrPh.top := FALSE;
	StrPh.error := FALSE;

	CASE act OF
		(*DualStateImAction.on*)   _on :im.inOpcCommandsDisabled:=TRUE;
                                                    im.inCommand_Alg := 1; (*cmd_open*)
		(*DualStateImAction.off*) _off :im.inOpcCommandsDisabled:=TRUE;
                                                    im.inCommand_Alg := 2; (*cmd_close*)
	END_CASE;
END_IF;

IF StrPh.start OR StrPh.reset THEN
    StrPh.run:=FALSE;
END_IF;

IF StrPh.start AND NOT StrPh.top THEN
                    CommandFault_Trig(CLK := im.CommandFault);
                    IF CommandFault_Trig.Q THEN
	          StrPh.error := TRUE;
                    END_IF;

		CASE act OF
		(*_DualStateImAction.on*)    _on: StrPh.top := im.onStatus = _statusDualInput.STATUS_ON;
		(*_DualStateImAction.off*)  _off: StrPh.top := im.onStatus = _statusDualInput.STATUS_OFF;
		END_CASE;

END_IF;

reset_Trig(CLK := StrPh.reset);
IF reset_Trig.Q THEN
	StrPh.start := FALSE;
	StrPh.error := FALSE;
	StrPh.top := FALSE;
          StrPh.reset:=FALSE;
END_IF;

StrPh.startStatus := SHL(BOOL_TO_DWORD(StrPh.start), PhaseNumber);
StrPh.errorStatus := SHL(BOOL_TO_DWORD(StrPh.error), PhaseNumber);
StrPh.topStatus := SHL(BOOL_TO_DWORD(StrPh.top), PhaseNumber);

(* ---- fb_ph_SectionSwitch.st ---- *)
FUNCTION_BLOCK fb_ph_SectionSwitch

VAR_IN_OUT
	im : struct_SectionSwitch;
END_VAR

VAR_INPUT
	act : TYPE_DualStateImAction;
	PhaseNumber : UINT;
END_VAR

VAR_IN_OUT
	StrPh : struct_PhaseAlgoritm;
END_VAR

VAR
	CommandFault_Trig : R_TRIG;
	reset_Trig : R_TRIG;
	_statusDualInput : TYPE_statusDualInput;
END_VAR

IF StrPh.run AND NOT StrPh.start THEN
	StrPh.start := TRUE;
	StrPh.top := FALSE;
	StrPh.error := FALSE;
          StrPh.run:=FALSE;

	CASE act OF
		(*DualStateImAction.on*)   _on : im.inOpcCommandsDisabled:=TRUE;
                                                     im.inCommand_Alg := 1; (*cmd_open*)
		(*DualStateImAction.off*) _off : im.inOpcCommandsDisabled:=TRUE;
                                                     im.inCommand_Alg := 2; (*cmd_close*)
	END_CASE;
END_IF;

IF StrPh.start AND NOT StrPh.top THEN
                    CommandFault_Trig(CLK := im.CommandFault);
                    IF CommandFault_Trig.Q THEN
	          StrPh.error := TRUE;
                    END_IF;

		CASE act OF
		(*_DualStateImAction.on*)    _on: StrPh.top := im.onStatus = _statusDualInput.STATUS_ON;
		(*_DualStateImAction.off*)  _off: StrPh.top := im.onStatus = _statusDualInput.STATUS_OFF;
		END_CASE;

END_IF;

IF StrPh.top THEN
StrPh.error := FALSE;
END_IF;

reset_Trig(CLK := StrPh.reset);
IF reset_Trig.Q THEN
	StrPh.start := FALSE;
	StrPh.error := FALSE;
	StrPh.top := FALSE;
          StrPh.run:=FALSE;
          StrPh.reset:=FALSE;
END_IF;

StrPh.startStatus := SHL(BOOL_TO_DWORD(StrPh.start), PhaseNumber);
StrPh.errorStatus := SHL(BOOL_TO_DWORD(StrPh.error), PhaseNumber);
StrPh.topStatus := SHL(BOOL_TO_DWORD(StrPh.top), PhaseNumber);

(* ---- fb_ph_Switch.st ---- *)
FUNCTION_BLOCK fb_ph_Switch

VAR_IN_OUT
	im : struct_Switch;
END_VAR

VAR_INPUT
	act : TYPE_DualStateImAction;
	PhaseNumber : UINT;
END_VAR

VAR_IN_OUT
	StrPh : struct_PhaseAlgoritm;
END_VAR

VAR
	CommandFault_Trig : R_TRIG;
	reset_Trig : R_TRIG;
	_statusDualInput : TYPE_statusDualInput;
END_VAR

IF StrPh.run AND NOT StrPh.start THEN
	StrPh.start := TRUE;
	StrPh.top := FALSE;
	StrPh.error := FALSE;
          StrPh.run:=FALSE;

	CASE act OF
		(*DualStateImAction.on*)   _on :im.inOpcCommandsDisabled:=TRUE;
                                                    im.inCommand_Alg := 1; (*cmd_open*)
		(*DualStateImAction.off*) _off :im.inOpcCommandsDisabled:=TRUE;
                                                    im.inCommand_Alg := 2; (*cmd_close*)
	END_CASE;
END_IF;

IF StrPh.start AND NOT StrPh.top THEN
                    CommandFault_Trig(CLK := im.CommandFault);
                    IF CommandFault_Trig.Q THEN
	          StrPh.error := TRUE;
                    END_IF;

		CASE act OF
		(*_DualStateImAction.on*)    _on: StrPh.top := im.onStatus = _statusDualInput.STATUS_ON;
		(*_DualStateImAction.off*)  _off: StrPh.top := im.onStatus = _statusDualInput.STATUS_OFF;
		END_CASE;

END_IF;

IF StrPh.top THEN
StrPh.error := FALSE;
END_IF;

reset_Trig(CLK := StrPh.reset);
IF reset_Trig.Q THEN
	StrPh.start := FALSE;
	StrPh.error := FALSE;
	StrPh.top := FALSE;
          StrPh.run:=FALSE;
          StrPh.reset:=FALSE;
END_IF;

StrPh.startStatus := SHL(BOOL_TO_DWORD(StrPh.start), PhaseNumber);
StrPh.errorStatus := SHL(BOOL_TO_DWORD(StrPh.error), PhaseNumber);
StrPh.topStatus := SHL(BOOL_TO_DWORD(StrPh.top), PhaseNumber);

(* ---- fb_ph_Timer.st ---- *)
FUNCTION_BLOCK fb_ph_Timer

VAR_INPUT
	delay : TIME;
	PhaseNumber : UINT;
END_VAR

VAR_IN_OUT
	StrPh : struct_PhaseAlgoritm;
END_VAR

VAR
	CommandFault_Trig : R_TRIG;
	reset_Trig : R_TRIG;
END_VAR

VAR_IN_OUT
	timer : UINT;
END_VAR

VAR
	_timer : TON;
	_statusDualInput : TYPE_statusDualInput;
END_VAR

IF StrPh.run AND NOT StrPh.start THEN
	StrPh.start := TRUE;
	StrPh.top := FALSE;
	StrPh.error := FALSE;
          StrPh.run:=FALSE;

END_IF;

_timer(IN:=StrPh.start, PT:=delay);

timer:=TIME_TO_UINT(delay -_timer.ET);

IF StrPh.start AND NOT StrPh.top THEN
StrPh.top:=_timer.Q;
END_IF;

reset_Trig(CLK := StrPh.reset);
IF reset_Trig.Q THEN
	StrPh.start := FALSE;
	StrPh.error := FALSE;
	StrPh.top := FALSE;
          StrPh.run:=FALSE;
          (*timer:=TIME_TO_UINT(delay -_timer.ET);*)
          StrPh.reset:=FALSE;
END_IF;

StrPh.startStatus := SHL(BOOL_TO_DWORD(StrPh.start), PhaseNumber);
StrPh.errorStatus := SHL(BOOL_TO_DWORD(StrPh.error), PhaseNumber);
StrPh.topStatus := SHL(BOOL_TO_DWORD(StrPh.top), PhaseNumber);

(* ---- fb_ph_WaitAnalogValue.st ---- *)
FUNCTION_BLOCK fb_ph_WaitAnalogValue

VAR_IN_OUT
	ai : struct_AI;
END_VAR

VAR_INPUT
	more : LREAL;
	less : LREAL;
	PhaseNumber : UINT;
END_VAR

VAR_IN_OUT
	StrPh : struct_PhaseAlgoritm;
END_VAR

VAR
	CommandFault_Trig : R_TRIG;
	reset_Trig : R_TRIG;
	_statusAi : TYPE_StatusAi;
	_statusDualInput : TYPE_statusDualInput;
END_VAR

IF StrPh.run AND NOT StrPh.start THEN
	StrPh.start := TRUE;
	StrPh.top := FALSE;
	StrPh.error := FALSE;
          StrPh.run:=FALSE;
END_IF;

IF StrPh.start AND NOT StrPh.top THEN
                    IF ai.interval < _statusAi.normal THEN
	              StrPh.error := TRUE;
                        StrPh.top:=FALSE;
                    ELSE
                            IF (more<>0.0) OR (less<>0.0) THEN
                            StrPh.top:=TRUE;
	                    IF more<>0.0 THEN StrPh.top:=StrPh.top AND (ai.value > more); END_IF;
	                    IF less<>0.0 THEN StrPh.top:=StrPh.top AND (ai.value < less); END_IF;
                            ELSE
	                  StrPh.top:=TRUE;
                            END_IF;
                   END_IF;
END_IF;

IF StrPh.top THEN
StrPh.error := FALSE;
END_IF;

reset_Trig(CLK := StrPh.reset);
IF reset_Trig.Q THEN
	StrPh.start := FALSE;
	StrPh.error := FALSE;
	StrPh.top := FALSE;
          StrPh.run:=FALSE;
          StrPh.reset:=FALSE;
END_IF;

StrPh.startStatus := SHL(BOOL_TO_DWORD(StrPh.start), PhaseNumber);
StrPh.errorStatus := SHL(BOOL_TO_DWORD(StrPh.error), PhaseNumber);
StrPh.topStatus := SHL(BOOL_TO_DWORD(StrPh.top), PhaseNumber);

(* ---- fb_ProtectionsManager.st ---- *)
FUNCTION_BLOCK fb_ProtectionsManager

VAR
	cmd : BYTE;
END_VAR

VAR_IN_OUT
	str_PM : struct_ProtectionsManager;
END_VAR

VAR
	lastCmd : BYTE;
	autoRunPriznak : BOOL;
	onInit : BOOL;
END_VAR

VAR_EXTERNAL
	protections : ProtectionsConfig;
END_VAR

VAR
	timerUnBlock : TON;
	timerAutoRun : TON;
	UnBlockPriznak : BOOL;
END_VAR

IF NOT onInit THEN

    autoRunProtections(protections);
onInit:=TRUE;
END_IF;

str_PM.protectionInRemont:=anyProtectioninRemont(protections);

cmd := str_PM.inCommand;

IF cmd <> 0 AND lastCmd <> cmd then
              UnBlockPriznak:=TRUE;
	CASE BYTE_TO_INT(cmd) OF

		(*RestartAllSignaling*) 1: 	ResetAllSignaling(protections);
				          autoRunPriznak:=TRUE;

	        (*RestartAllProtections*) 2: 	ResetAllProtections(protections);
                                                  autoRunPriznak:=TRUE;

                      (*CheckProtections*)  3: 	RunAllProtections(protections);

	         (*ResetAllProtections*)  4: 	ResetAllProtections(protections);

	END_CASE;

END_IF;
lastCmd := cmd;
timerUnBlock(IN:=UnBlockPriznak, PT:=T#1S);
timerAutoRun(IN:=autoRunPriznak, PT:=T#500MS);

IF timerAutoRun.Q THEN autoRunProtections(protections);
END_IF;

IF timerUnBlock.Q THEN
lastCmd:= 0;
str_PM.inCommand:=0;
autoRunPriznak:=FALSE;
UnBlockPriznak:=FALSE;
END_IF;

(* ---- fb_puskOilSystemAlg.st ---- *)
FUNCTION_BLOCK fb_puskOilSystemAlg

VAR_IN_OUT
	StrAlg : struct_Alg;
END_VAR

VAR
	pnsOn : struct_PhaseAlgoritm;
	LowOil : struct_PhaseAlgoritm;
	BreakPuskTimer_Poil : struct_PhaseAlgoritm;
	Poil_DefenseActive : struct_PhaseAlgoritm;
	autoNuOn : struct_PhaseAlgoritm;
	nuOn : struct_PhaseAlgoritm;
	nu1On : struct_PhaseAlgoritm;
	nu2On : struct_PhaseAlgoritm;
	di_dPmg : struct_PhaseAlgoritm;
	dP_oilGas100 : struct_PhaseAlgoritm;
	runProtect_dP : struct_PhaseAlgoritm;
	testUnsuccessful : struct_PhaseAlgoritm;
	fb_pnsOn : fb_ph_Switch;
	fb_LowOil : fb_ph_WaitAnalogValue;
	fb_BreakPuskTimer_Poil : fb_ph_Timer;
	fb_Poil_DefenseActive : fb_ph_CustomPhase;
	fb_nuOn : fb_ph_CustomPhase;
	fb_nu1On : fb_ph_OilPump;
	fb_nu2On : fb_ph_OilPump;
	fb_autoNuOn : fb_ph_algoritm;
	fb_di_dPmg : fb_ph_CustomPhase;
	fb_dP_oilGas100 : fb_ph_WaitAnalogValue;
	fb_runProtect_dP : fb_ph_CustomPhase;
	fb_testUnsuccessful : fb_ph_CustomPhase;
	_sunpackerCommand : fb_sunpackerCommand;
	_statusAi : TYPE_StatusAi;
	_Answers : TYPE_Answers;
	_statusDualInput : TYPE_statusDualInput;
	_DualStateImAction : TYPE_DualStateImAction;
	_PhaseAlgoritmAction : TYPE_PhaseAlgoritmAction;
	source : BYTE;
	cmd : BYTE;
	lastCmd : BYTE;
	source_for_Status : BYTE;
	cmd_for_Status : BYTE;
	command_error_for_Status : BYTE;
	resetCmdTimer : TON;
	resetCmdTimerPriznak : BOOL;
	onInit : BOOL;
	waitReset : TON;
END_VAR

VAR_EXTERNAL
	IM : ImConfig;
	algoritms : AlgoritmsConfig;
	ai : AiConfig;
	protections : ProtectionsConfig;
	AlgTimers : struct_AlgTimers;
END_VAR

IF NOT onInit THEN
               fb_pnsOn(phaseNumber:=0, act:=_on);
              fb_LowOil(phaseNumber:=1);
 fb_BreakPuskTimer_Poil(phaseNumber:=3, delay:=T#240S);
  fb_Poil_DefenseActive(phaseNumber:=5);
                fb_nuOn(phaseNumber:=6);
               fb_nu1On(phaseNumber:=11, act:=_on);
               fb_nu2On(phaseNumber:=12, act:=_on);
            fb_autoNuOn(phaseNumber:=7, act:=_run, waitCompletion:=FALSE);
             fb_di_dPmg(phaseNumber:=8);
        fb_dP_oilGas100(phaseNumber:=9);
       fb_runProtect_dP(phaseNumber:=10);
    fb_testUnsuccessful(phaseNumber:=17);

onInit:=TRUE;
END_IF;

              fb_pnsOn(StrPh:=pnsOn, Im:=IM.pns);
             (*fb_LowOil(StrPh:=LowOil, ai:=ai.Pmasla_posle_GNS, more:=im.AutoPns_UstRun.Value);*)
fb_BreakPuskTimer_Poil(StrPh:=BreakPuskTimer_Poil, timer:=AlgTimers.puskOilSystem_BreakPuskTimer_Poil);
 fb_Poil_DefenseActive(StrPh:=Poil_DefenseActive);
               fb_nuOn(StrPh:=nuOn);
              fb_nu1On(StrPh:=nu1On, Im:=Im.nu1);
              fb_nu2On(StrPh:=nu2On, Im:=Im.nu2);
           fb_autoNuOn(StrPh:=autoNuOn, alg:=algoritms.autoNu);
            fb_di_dPmg(StrPh:=di_dPmg);
       (*fb_dP_oilGas100(StrPh:=dP_oilGas100, ai:=ai.Tmasla_MB, more:=im.PuskOilSystem_UstdPmg.Value);*)
      fb_runProtect_dP(StrPh:=runProtect_dP);
   fb_testUnsuccessful(StrPh:=testUnsuccessful);

IF StrAlg.isRuning THEN

    StrAlg.hasError := LowOil.error OR dP_oilGas100.error OR pnsOn.error OR testUnsuccessful.error;

    IF pnsOn.top THEN
        runPhase(LowOil);
    END_IF;

    IF LowOil.top THEN
        runAiProtection(protections.Os_sdvig_nagnetatelja_minus);
        (*runDiProtection(protections.Vibro_skorost_OP_shesterni_RED_T6);*)
        runPhase(Poil_DefenseActive);
        (*IM.SingleSignals.P_oil_low.Disabled_Sig:=FALSE;*)
        ai.Pmasla_posle_GNS.Disabled_LA:=FALSE;
        ai.Pmasla_posle_GNS.Disabled_LW:=FALSE;
        ai.Pmasla_posle_NU.Disabled_LW:=FALSE;
    END_IF;

    IF Poil_DefenseActive.start AND NOT Poil_DefenseActive.top THEN
       Poil_DefenseActive.top:=protections.Os_sdvig_nagnetatelja_minus.isRunning AND protections.Vibro_skorost_OP_shesterni_RED_T6.isRunning;
    END_IF;

    IF Poil_DefenseActive.top THEN
       (* runPhase(autoNuOn);*)
	runPhase(nuOn);
    END_IF;

    IF nuOn.start AND NOT nuOn.top THEN
       (* IF IM.SingleOutputs.Value = 0 THEN
            runPhase(nu1On);
        END_IF;

        IF IM.SingleOutputs.Value = 1 THEN
            runPhase(nu2On);
        END_IF;*)
       nuOn.top:= Im.nu1.onStatus = _statusDualInput.STATUS_ON OR Im.nu2.onStatus = _statusDualInput.STATUS_ON;
    END_IF;

    IF nuOn.top THEN
	runPhase(di_dPmg);
          runPhase(dP_oilGas100);
    END_IF;

    (*IF di_dPmg.start AND NOT di_dPmg.top THEN
       di_dPmg.top:= NOT IM.SingleSignals.dP_oilgaz_low.Q;
    END_IF;*)

    IF dP_oilGas100.top AND di_dPmg.top THEN
          runPhase(autoNuOn);
	runPhase(runProtect_dP);
	runAiProtection(protections.Os_sdvig_nagnetatelja_plus);
          (*runDiProtection(protections.Vibro_skorost_OP_shesterni_RED_T5);
          IM.SingleSignals.dP_oilgaz_low.Disabled_Sig:=FALSE;
          ai.Tmasla_MB.Disabled_LA:=FALSE;
          ai.Tmasla_MB.Disabled_LW:=FALSE;*)
    END_IF;

    IF runProtect_dP.start AND NOT runProtect_dP.top THEN
       runProtect_dP.top:= protections.Os_sdvig_nagnetatelja_plus.isRunning AND protections.Vibro_skorost_OP_shesterni_RED_T5.isRunning;
    END_IF;

    IF BreakPuskTimer_Poil.top AND (NOT runProtect_dP.top) THEN
	testUnsuccessful.error:=TRUE;
    END_IF;

    IF runProtect_dP.top THEN
          resetPhase(BreakPuskTimer_Poil);
	waitReset(IN:=TRUE);
    END_IF;

    IF waitReset.Q AND NOT (algoritms.Apusk.isRuning OR algoritms.SemiAutoPusk.isRuning) THEN
    resetAndDisable(StrAlg);
    END_IF;

    StrAlg.isEnded:=runProtect_dP.top;
END_IF;

StrAlg.CanRun := StrAlg.inCanRun;
StrAlg.OpcCommandsDisabled := StrAlg.inOpcCommandsDisabled;

(* ---- Если управление с ВУ заблокировано, то  передаем команду из алгоритма ---- *)
IF StrAlg.inOpcCommandsDisabled THEN
	StrAlg.inCommand := StrAlg.inCommand_Alg;
ELSE (* иначе передаем команду с АРМа*)
	StrAlg.inCommand := StrAlg.inCommand_ARM;
END_IF;

_sunpackerCommand(command := StrAlg.inCommand);
	source := _sunpackerCommand.source;
	cmd := _sunpackerCommand.cmd;

IF cmd <> 0 AND lastCmd <> cmd AND (((NOT StrAlg.opcCommandsDisabled) AND source > 0) OR source = 0) then
	CASE BYTE_TO_INT(cmd) OF
		(*cmdRun*) 1: 	IF (StrAlg.CanRun) THEN
					StrAlg.isRuning := TRUE;
					StrAlg.isEnded := FALSE;
					StrAlg.hasError := FALSE;
					(*****************       OnRun       *****************)
                                                  runPhase(pnsOn);
                                                  runPhase(BreakPuskTimer_Poil);
                                                  runPhase(testUnsuccessful);
					cmd_for_Status := cmd;
					source_for_Status := source;
					command_error_for_Status := 0;
				ELSE
					StrAlg.isRuning := FALSE;
					StrAlg.isEnded := FALSE;
					StrAlg.hasError 	:= FALSE;

					cmd_for_Status := 0;
					source_for_Status := source;
					command_error_for_Status := cmd;
				END_IF;
		(*cmdReset*) 2: 	StrAlg.isRuning := FALSE;
				StrAlg.isEnded := FALSE;
				StrAlg.hasError 	:= FALSE;

                                         (*****************       OnReset       *****************)
                                        waitReset(IN:=FALSE);
                                        resetPhase(pnsOn);
                                        resetPhase(LowOil);
                                        resetPhase(BreakPuskTimer_Poil);
                                        resetPhase(Poil_DefenseActive);
                                        resetPhase(autoNuOn);
                                        resetPhase(nu1On);
                                        resetPhase(nu2On);
                                        resetPhase(nuOn);
                                        resetPhase(di_dPmg);
                                        resetPhase(dP_oilGas100);
                                        resetPhase(runProtect_dP);
                                        resetPhase(testUnsuccessful);
	                              (*protections.Os_sdvig_nagnetatelja_minus.inOpcCommandsDisabled:=FALSE;
                                        protections.Vibro_skorost_OP_shesterni_RED_T6.inOpcCommandsDisabled:=FALSE;
                                        protections.Os_sdvig_nagnetatelja_plus.inOpcCommandsDisabled:=FALSE;
                                        protections.Vibro_skorost_OP_shesterni_RED_T5.inOpcCommandsDisabled:=FALSE;*)

				cmd_for_Status := cmd;
				source_for_Status := source;
				command_error_for_Status := 0;
	END_CASE;
	resetCmdTimer(IN := false);
	resetCmdTimerPriznak := TRUE;
END_IF;
lastCmd := cmd;

resetCmdTimer(IN := resetCmdTimerPriznak, PT := T#5S);
IF resetCmdTimer.Q THEN
	resetCmdTimerPriznak := FALSE;
	source_for_Status := 0;
	cmd_for_Status := 0;
	command_error_for_Status := 0;
END_IF;

StrAlg.Start:= pnsOn.startStatus
            OR LowOil.startStatus
            OR BreakPuskTimer_Poil.startStatus
            OR Poil_DefenseActive.startStatus
            OR nuOn.startStatus
            OR di_dPmg.startStatus
            OR dP_oilGas100.startStatus
            OR runProtect_dP.startStatus
            OR testUnsuccessful.startStatus;

StrAlg.Error:= pnsOn.errorStatus
            OR LowOil.errorStatus
            OR BreakPuskTimer_Poil.errorStatus
            OR Poil_DefenseActive.errorStatus
            OR nuOn.errorStatus
            OR di_dPmg.errorStatus
            OR dP_oilGas100.errorStatus
            OR runProtect_dP.errorStatus
            OR testUnsuccessful.errorStatus;

StrAlg.Top:=   pnsOn.topStatus
            OR LowOil.topStatus
            OR BreakPuskTimer_Poil.topStatus
            OR Poil_DefenseActive.topStatus
            OR nuOn.topStatus
            OR di_dPmg.topStatus
            OR dP_oilGas100.topStatus
            OR runProtect_dP.topStatus
            OR testUnsuccessful.topStatus;

(*TODO: TYPE PROGRAM CODE HERE*)
StrAlg.status :=  SHL(BYTE_TO_DWORD(source_for_Status), 29)
			OR SHL(BYTE_TO_DWORD(cmd_for_Status), 26)
			OR SHL(BYTE_TO_DWORD(command_error_for_Status), 23)
			OR SHL(BOOL_TO_DWORD(StrAlg.OpcCommandsDisabled ), 21)
			OR SHL(BOOL_TO_DWORD(StrAlg.hasError),4)
			OR SHL(BOOL_TO_DWORD(StrAlg.CanRun),2)
			OR SHL(BOOL_TO_DWORD(StrAlg.isEnded),1)
			OR BOOL_TO_DWORD(StrAlg.isRuning);

(* ---- fb_Question.st ---- *)
FUNCTION_BLOCK fb_Question

VAR_IN_OUT
	StrQ : struct_Question;
END_VAR

VAR
	Asked : UINT;
	_answers : TYPE_Answers;
	_sunpackerCommand : fb_sunpackerCommand;
	source : BYTE;
	parametr : BYTE;
	lastParametr : BYTE;
	cmd : BYTE;
	source_for_Status : BYTE;
	cmd_for_Status : BYTE;
	command_error_for_Status : BYTE;
	resetCmdTimer : TON;
	resetCmdTimerPriznak : BOOL;
	reset_Trig : R_TRIG;
END_VAR

VAR CONSTANT
	cmd_answer : UINT          := 1;
END_VAR

StrQ.OpcCommandsDisabled := StrQ.inopcCommandsDisabled;

IF StrQ.ask THEN
StrQ.inopcCommandsDisabled:=FALSE;
    IF Asked=0 THEN
	Asked:=StrQ.AnswerVariants;
	StrQ.answer:=_answers.ANS_NONE;
    END_IF;

    _sunpackerCommand(command := StrQ.inCommand);
	source := _sunpackerCommand.source;
          parametr := _sunpackerCommand.parametr;
	cmd := _sunpackerCommand.cmd;

    IF cmd <> 0 AND lastParametr <> parametr AND ((NOT StrQ.OpcCommandsDisabled) AND source > 0)  then
	CASE BYTE_TO_INT(cmd) OF
	                               1 :

				IF Asked<>0 THEN
                                           (* CASE BYTE_TO_INT(parametr) OF
                                            1: answer:=_answers.ANS_YES;
                                            2: answer:=_answers.ANS_NO;
                                            4: answer:=_answers.ANS_CANCEL;
                                            8: answer:=_answers.ANS_RETRY;
	                                  END_CASE;*)
                                        StrQ.answer:=BYTE_TO_UINT(parametr);
                                        command_error_for_Status := 0;
                                        ELSE
	                              command_error_for_Status := cmd;
                                        END_IF;
	END_CASE;
	source_for_Status := source;
	cmd_for_Status := cmd;
	resetCmdTimer(IN := FALSE);
	resetCmdTimerPriznak := TRUE;
    END_IF;

    lastParametr := parametr;

    resetCmdTimer(IN := resetCmdTimerPriznak, PT := T#5S);
    IF resetCmdTimer.Q THEN
	resetCmdTimerPriznak := FALSE;
	source_for_Status := 0;
	cmd_for_Status := 0;
	command_error_for_Status := 0;
    END_IF;
END_IF;

reset_Trig(CLK := StrQ.reset);
IF reset_Trig.Q THEN
	Asked:=0;
	StrQ.answer:=0;
          StrQ.ask:=FALSE;
          StrQ.reset:=FALSE;
	StrQ.inopcCommandsDisabled:=TRUE;
END_IF;

StrQ.status := SHL(BYTE_TO_DWORD(source_for_Status), 29)
			OR SHL(BYTE_TO_DWORD(cmd_for_Status), 26)
			OR SHL(BYTE_TO_DWORD(command_error_for_Status), 23)
			OR SHL(BOOL_TO_DWORD(StrQ.OpcCommandsDisabled ), 21);
IF StrQ.answer = 0 THEN
    StrQ.status := StrQ.status  OR SHL(UINT_TO_DWORD(asked), 6);
ELSE
    StrQ.status := StrQ.status  OR SHL(UINT_TO_DWORD(StrQ.answer), 6);
END_IF;

(* ---- fb_RashodAlg.st ---- *)
FUNCTION_BLOCK fb_RashodAlg

VAR_INPUT
	P_gasIn : struct_AI;
END_VAR

VAR_IN_OUT
	StrAi : struct_AI;
END_VAR

VAR_INPUT
	T_gasIn : struct_AI;
	dP_konf : struct_AI;
	K : struct_AnalogParametr;
	A : struct_AnalogParametr;
	y0 : struct_AnalogParametr;
END_VAR

VAR
	num : LREAL;
	den : LREAL;
	_statusAi : TYPE_StatusAi;
END_VAR

VAR CONSTANT
	P0 : LREAL          := 0.1033;
	T0 : LREAL          := 293.0;
END_VAR

strAI.opcCommandsDisabled := strAI.inopcCommandsDisabled ;

IF (P_gasIn.interval < _statusAi.normal) OR
   (T_gasIn.interval < _statusAi.normal) OR
   (dP_konf.interval < _statusAi.normal) THEN
	StrAi.interval := _statusAi.NOTRELIABLE;
          strAI.status := 	SHL(BOOL_TO_DWORD(strAI.OpcCommandsDisabled ), 21)
	OR BYTE_TO_DWORD(strAI.interval);
	RETURN;
END_IF;

IF (P_gasIn.value <0.3) THEN
	StrAi.interval := _statusAi.normal;
	StrAi.value:= 0.0;
          strAI.status := 	SHL(BOOL_TO_DWORD(strAI.OpcCommandsDisabled ), 21)
	OR BYTE_TO_DWORD(strAI.interval);
	RETURN;
END_IF;

StrAi.interval:= _statusAi.normal;

num:= (dP_konf.Value/1000.0)*(T_gasIn.value+273.0)*P0*735.56*K.Value;
den:= y0.Value*P_gasIn.value*T0 ;

StrAi.value:= A.Value*SQRT(num/den);

strAI.status := 	SHL(BOOL_TO_DWORD(strAI.OpcCommandsDisabled ), 21) (* Управление в ВУ заблокировано *)
		OR BYTE_TO_DWORD(strAI.interval);	              (* интервал *)

(* ---- fb_SectionSwitch.st ---- *)
FUNCTION_BLOCK fb_SectionSwitch

VAR_INPUT
	statOn : BOOL;
	statOff : BOOL;
	statOn_reliability : BOOL;
	statOff_reliability : BOOL;
END_VAR

VAR_IN_OUT
	StrSw : struct_SectionSwitch;
END_VAR

VAR_INPUT
	basketRolledIn : TYPE_ReliableBit;
	basketRolledOut : TYPE_ReliableBit;
	basketTest : TYPE_ReliableBit;
	inNs : TYPE_ReliableBit;
	inoffKNA : TYPE_ReliableBit;
	inAccident : TYPE_ReliableBit;
	inLocal : TYPE_ReliableBit;
	inDistance : TYPE_ReliableBit;
	inBreakCmdOn : TYPE_ReliableBit;
	inBreakCmdOff : TYPE_ReliableBit;
END_VAR

VAR
	onInit : BOOL          := FALSE;
	_statOn : BOOL;
	_statOff : BOOL;
	getSdvig : BOOL;
	lastOnStatus : BYTE;
	cmd : BYTE;
	source : BYTE;
	lastCmd : BYTE;
	source_for_Status : BYTE;
	cmd_for_Status : BYTE;
	command_error_for_Status : BYTE;
	_basketRolledIn : TYPE_ReliableBit;
	_basketRolledOut : TYPE_ReliableBit;
	_basketTest : TYPE_ReliableBit;
	_sunpackerCommand : fb_sunpackerCommand;
	_statusDualInput : TYPE_statusDualInput;
	_statusBasket : TYPE_basketStats;
	_commandDualInput : TYPE_commandDualInput;
	_commandErrorTimer : BOOL;
	resetErrorTimer : BOOL;
	_changWithoutCommand : BOOL;
	errorCMDTimer : TON;
	_errorReset : TON;
	sdvigReset : TON;
	outputsSets : TOF;
END_VAR

VAR_IN_OUT
	cmdOn : BOOL;
	cmdOff : BOOL;
END_VAR

IF NOT onInit THEN
IF StrSw.ISVALIDREF_cmdOn XOR StrSw.ISVALIDREF_cmdOff THEN
	IF 	StrSw.ISVALIDREF_cmdOn THEN
		lastCmd:= 2; (*baseCmdOff*)
	ELSE
		lastCmd:= 1; (*baseCmdOn*)
	END_IF;
END_IF;
onInit:=TRUE;
END_IF;

(* ---- Формирование состояния тележки ---- *)

IF (NOT StrSw.ISVALIDREF_basketRolledIn) AND (NOT StrSw.ISVALIDREF_basketRolledOut) THEN
          StrSw.basketStatus:=_statusBasket.BASKET_NOTDEFINED;
ELSE
		IF StrSw.ISVALIDREF_basketTest THEN
		_basketTest:=basketTest;
	ELSE
		_basketTest.reliability:=TRUE;
		_basketTest.value :=FALSE;
	END_IF;

	IF StrSw.ISVALIDREF_basketRolledIn THEN
		_basketRolledIn:=basketRolledIn;
	ELSE
		_basketRolledIn:=basketRolledOut;
		IF StrSw.ISVALIDREF_basketTest THEN
		_basketRolledIn.value:=NOT (_basketRolledIn.value OR _basketTest.value);
		ELSE
		_basketRolledIn.value:= NOT _basketRolledIn.value;
		END_IF;

	END_IF;

	IF StrSw.ISVALIDREF_basketRolledOut THEN
		_basketRolledOut:=basketRolledOut;
	ELSE
		_basketRolledOut:=basketRolledIn;
		IF StrSw.ISVALIDREF_basketTest THEN
		_basketRolledOut.value:= NOT (_basketRolledOut.value OR _basketTest.value );
		ELSE
			_basketRolledOut.value := NOT _basketRolledout.value;
		END_IF;

	END_IF;

IF _basketRolledIn.reliability AND _basketRolledOut.reliability AND _basketTest.reliability THEN
		IF (BOOL_TO_INT(_basketRolledIn.value)+BOOL_TO_INT(_basketRolledOut.value)+BOOL_TO_INT(_basketTest.value))=1 THEN
			IF _basketRolledIn.value THEN
				StrSw.basketStatus:=_statusBasket.BASKET_ROLLEDIN;
			ELSIF _basketRolledOut.value THEN
				StrSw.basketStatus:=_statusBasket.BASKET_ROLLEDOUT;
			ELSIF _basketTest.value THEN
				StrSw.basketStatus:=_statusBasket.BASKET_TEST;
			END_IF;
		ELSE
			StrSw.basketStatus:=_statusBasket.BASKET_ERROR;
		END_IF;
	ELSE
		StrSw.basketStatus:=_statusBasket.BASKET_NOTDEFINED;
	END_IF;
END_IF;

(* ---- Если управление с ВУ заблокировано, то в ИМ передаем команду из алгоритма ---- *)
IF StrSw.inOpcCommandsDisabled THEN
	StrSw.inCommand := StrSw.inCommand_Alg;
ELSE (* иначе передаем команду с АРМа*)
	StrSw.inCommand := StrSw.inCommand_ARM;
END_IF;

(* ---- Формирование состояния механизма ---- *)

IF (StrSw.ISVALIDREF_statOn) OR (StrSw.ISVALIDREF_statOff) THEN
	IF (StrSw.ISVALIDREF_statOn) AND (StrSw.ISVALIDREF_statOff) THEN
	StrSw.reliability:= statOn_reliability AND statOff_reliability;
		_statOn  := statOn;
		_statOff := statOff;
	ELSIF (StrSw.ISVALIDREF_statOn) THEN
                     StrSw.reliability:= statOn_reliability;
		_statOn  := statOn;
		_statOff := NOT statOn;
	ELSIF (StrSw.ISVALIDREF_statOff) THEN
		 StrSw.reliability:= statOff_reliability;
		_statOn  := NOT statOff;
		_statOff :=statOff;
	END_IF;

	IF StrSw.reliability THEN
		IF _statOn AND NOT _statOff 		THEN 	StrSw.onStatus := _statusDualInput.STATUS_ON;
		ELSIF _statOff AND NOT _statOn 	THEN 	StrSw.onStatus := _statusDualInput.Status_OFF;
		ELSIF NOT _statOn AND NOT _statOff 	THEN 	StrSw.onStatus := _statusDualInput.STATUS_TRANSITIONAL;
		ELSE					StrSw.onStatus := _statusDualInput.STATUS_ERROR;
                    END_IF;

	ELSE
		StrSw.onStatus := _statusDualInput.STATUS_NOTDEFINED;

	END_IF;
ELSE
	CASE BYTE_TO_INT(lastCmd) OF
		(*baseCmdOn*) 1: StrSw.onStatus  := _statusDualInput.STATUS_ON;
		(*baseCmdOff*) 2: StrSw.onStatus  := _statusDualInput.STATUS_OFF;

	ELSE
		 StrSw.onStatus := _statusDualInput.STATUS_NOTDEFINED;

	END_CASE;
END_IF;

StrSw.Accident := inAccident.value AND inAccident.reliability;
StrSw.Ns := inNs.value AND inNs.reliability;
StrSw.Local := inLocal.value AND inLocal.reliability;
StrSw.Distance := inDistance.value AND inDistance.reliability;
StrSw.OpcCommandsDisabled := StrSw.inOpcCommandsDisabled;
StrSw.offKNA := inoffKNA.value AND inoffKNA.reliability;

(* ---- Формирование признака сдвига ---- *)

getSdvig := FALSE;
IF (StrSw.ISVALIDREF_cmdOn OR StrSw.ISVALIDREF_cmdOff) AND NOT StrSw.Local THEN
	IF NOT (StrSw.CmdOn OR StrSw.CmdOff) THEN
                     IF (lastOnStatus <> StrSw.onStatus AND
		(StrSw.onStatus <> _statusDualInput.STATUS_NOTDEFINED AND
                     StrSw.onStatus <> _statusDualInput.STATUS_ERROR)     AND
		(lastOnStatus <> _statusDualInput.STATUS_NOTDEFINED   AND
                     lastOnStatus <> _statusDualInput.STATUS_ERROR))
                    THEN
			getSdvig   := TRUE;
		END_IF;
	END_IF;
END_IF;

IF getSdvig THEN StrSw.sdvig:= TRUE; END_IF;

sdvigReset(IN:=StrSw.sdvig, PT:=T#15S);

IF sdvigReset.Q THEN StrSw.sdvig:=FALSE; END_IF;

lastOnStatus := StrSw.onStatus;
